// TIA Portal project "EMS" (V14)

(* hardware
DEVICE "S7-1200 station_2"  S7-1200 Station
   slot 0: "Rack_0"  S7-1200 Rack  Rack  V1.0
   slot 1: "EnergyManagement"  CPU 1211C AC/DC/Rly  6ES7 211-1BE40-0XB0  V4.2
   slot 101: "CM 1241 (RS422/485)_1"  6ES7 241-1CH32-0XB0  V2.2
*)

// ===== PLC "EnergyManagement"  CPU 1211C AC/DC/Rly =====

VAR_GLOBAL   // PLC tag table "Default tag table"
   "System_Byte" AT %MB1 : Byte;
   "FirstScan" AT %M1.0 : Bool;
   "DiagStatusUpdate" AT %M1.1 : Bool;
   "AlwaysTRUE" AT %M1.2 : Bool;
   "AlwaysFALSE" AT %M1.3 : Bool;
   "Clock_Byte" AT %MB0 : Byte;
   "Clock_10Hz" AT %M0.0 : Bool;
   "Clock_5Hz" AT %M0.1 : Bool;
   "Clock_2.5Hz" AT %M0.2 : Bool;
   "Clock_2Hz" AT %M0.3 : Bool;
   "Clock_1.25Hz" AT %M0.4 : Bool;
   "Clock_1Hz" AT %M0.5 : Bool;
   "Clock_0.625Hz" AT %M0.6 : Bool;
   "Clock_0.5Hz" AT %M0.7 : Bool;
   "Tag_1" AT %MB3 : Byte;
   "Tag_2" AT %M4.0 : Bool;
   "Tag_3" AT %M4.1 : Bool;
   "Tag_4" AT %M4.3 : Bool;
   "Tag_5" AT %M4.2 : Bool;
   "Tag_6" AT %MW102 : Word;
   "Tag_7" AT %M2.0 : Bool;
   "Tag_8" AT %M3.1 : Bool;
   "Tag_9" AT %MW10 : Word;
   "Tag_10" AT %MW100 : Word;
   "Tag_11" AT %M3.0 : Bool;
   "g" AT %M4.4 : Bool;
END_VAR

VAR_GLOBAL   // PLC tag table "GTL"
   "reteaOut" AT %Q0.0 : Bool;
   "baterieOut" AT %Q0.1 : Bool;
   "SPARE_OUT" AT %Q0.2 : Bool;
   "SPARE_OUT(1)" AT %Q0.3 : Bool;
   "stare" AT %I0.0 : Bool;
   "manual" AT %I0.2 : Bool;
   "retea" AT %I0.3 : Bool;
   "baterie" AT %I0.4 : Bool;
   "directieAuto" AT %I0.5 : Bool;   // FALSE - IntervalOrar TRUE - Piata
   "I1" AT %IW64 : Int;
   "I2" AT %IW66 : Int;
   "auto" AT %I0.1 : Bool;
END_VAR

VAR_GLOBAL CONSTANT   // PLC tag table "GTL"
   "Verificare" : Bool := 0;
END_VAR

TYPE "Modbus_Data"
   STRUCT
      Modbus : Struct
         Holding_Register : Struct
            Read : "UDT_DATA_PTR";
            Write : "UDT_DATA_PTR";
         END_STRUCT;
      END_STRUCT;
   END_STRUCT;
END_TYPE

TYPE "UDT_DATA_PTR"
   STRUCT
      DATA : Array[1..50] of Word;
   END_STRUCT;
END_TYPE

TYPE "UDT_MB_COMM_LOAD"
   STRUCT
      DONE : Bool;
      ERROR : Bool;
      STATUS : Word;
      ERROR_STATUS : Word;
   END_STRUCT;
END_TYPE

TYPE "Modbus_Slave_Data"
   STRUCT
      NDR : Bool;
      DR : Bool;
      ERROR : Bool;
      STATUS : Word;
      ERROR_STATUS : Word;
      MB_ADDR : UInt;
   END_STRUCT;
END_TYPE

TYPE "Modbus_M aster_Data"
   STRUCT
      DONE : Bool;
      BUSY : Bool;
      ERROR : Bool;
      STATUS : Word;
   END_STRUCT;
END_TYPE

DATA_BLOCK "GVL"   // DB3
{ S7_Optimized_Access := 'TRUE' }
VERSION : 0.1
   VAR
      "STEP" : Array[0..8] of Bool;
      MB_STEP : Array[0..8] of Bool;
   END_VAR
BEGIN
   "STEP"[0] := true;
   MB_STEP[0] := true;
END_DATA_BLOCK

DATA_BLOCK "IntervalOrar"   // DB6
{ S7_Optimized_Access := 'TRUE' }
VERSION : 0.1
   VAR
      "Error Code" : Word;
      OraCurenta : DTL;
      InceputProgram : DTL := DTL#1970-01-01-06:00:00;
      SfarsitProgram : DTL := DTL#1970-01-01-17:00:00;
   END_VAR
BEGIN
END_DATA_BLOCK

DATA_BLOCK "Piata"   // DB11
{ S7_Optimized_Access := 'TRUE' }
VERSION : 0.1
   VAR
      Prag : Int := 500;
      PretPiata : Int := 400;
   END_VAR
BEGIN
END_DATA_BLOCK

DATA_BLOCK "MB_Config"   // DB17
{ S7_Optimized_Access := 'FALSE' }
VERSION : 0.1
   VAR
      Modbus_Data : Struct
         DATA : Array[0..9] of UInt;
      END_STRUCT;
      Modbus_Data_1 : Struct
         DATA : Array[0..20] of Bool;
      END_STRUCT;
      Modbus_Slave : "Modbus_Slave_Data";
      MB_COMM_LOAD : "UDT_MB_COMM_LOAD";
      Modbus_Master : "Modbus_M aster_Data";
   END_VAR
BEGIN
   Modbus_Slave.MB_ADDR := 2;
   Modbus_Data.DATA[0] := 1;
   Modbus_Data.DATA[1] := 2;
   Modbus_Data.DATA[2] := 3;
   Modbus_Data.DATA[3] := 4;
   Modbus_Data.DATA[4] := 5;
   Modbus_Data.DATA[5] := 6;
   Modbus_Data.DATA[6] := 7;
   Modbus_Data.DATA[7] := 8;
   Modbus_Data.DATA[8] := 9;
END_DATA_BLOCK

DATA_BLOCK "ModBus_Commands"   // DB20
{ S7_Optimized_Access := 'FALSE' }
VERSION : 0.1
   VAR
      VERIF_REQUEST : Struct
         DATA : Array[1..8] of Byte;
      END_STRUCT;
      RESET_REQUEST : Struct
         DATA : Array[1..8] of Byte;
      END_STRUCT;
      SET_RETEA_ON : Struct   // DE VERIFICAT!! 42044
         DATA : Array[1..8] of Byte;
      END_STRUCT;
      SET_RETEA_OFF : Struct   // DE VERIFICAT!! 42044
         DATA : Array[1..8] of Byte;   // DE VERIFICAT!!
      END_STRUCT;
      SET_STARE_ON : Struct   // DE VERIFICAT!! 40200
         DATA : Array[1..8] of Byte;
      END_STRUCT;
      SET_STARE_OFF : Struct   // DE VERIFICAT!! 40200
         DATA : Array[1..8] of Byte;
      END_STRUCT;
      GET_CURR_HOUR_YIELD : Struct
         DATA : Array[1..8] of Byte;
      END_STRUCT;
      GET_CURR_DAY_YIELD : Struct
         DATA : Array[1..8] of Byte;
      END_STRUCT;
      GET_CURR_MONTH_YIELD : Struct
         DATA : Array[1..8] of Byte;
      END_STRUCT;
      GET_POWER_DIRECTION : Struct
         DATA : Array[1..8] of Byte;
      END_STRUCT;
      GET_DEVICE_STATUS : Struct
         DATA : Array[1..8] of Byte;
      END_STRUCT;
      PLACE_HOLDER : Struct
         DATA : Array[1..8] of Byte;
      END_STRUCT;
   END_VAR
BEGIN
   SET_RETEA_ON.DATA[8] := 16#68;
   SET_RETEA_ON.DATA[7] := 16#26;
   SET_RETEA_ON.DATA[6] := 16#01;
   SET_RETEA_ON.DATA[5] := 16#00;
   SET_RETEA_ON.DATA[4] := 16#34;
   SET_RETEA_ON.DATA[3] := 16#9D;
   SET_RETEA_ON.DATA[2] := 16#06;
   SET_RETEA_ON.DATA[1] := 16#01;
   SET_STARE_ON.DATA[8] := 16#64;
   SET_STARE_ON.DATA[7] := 16#E6;
   SET_STARE_ON.DATA[6] := 16#01;
   SET_STARE_ON.DATA[5] := 16#00;
   SET_STARE_ON.DATA[4] := 16#08;
   SET_STARE_ON.DATA[3] := 16#9D;
   SET_STARE_ON.DATA[2] := 16#06;
   SET_STARE_ON.DATA[1] := 16#01;
   RESET_REQUEST.DATA[1] := 16#FF;
   RESET_REQUEST.DATA[2] := 16#FF;
   RESET_REQUEST.DATA[3] := 16#FF;
   RESET_REQUEST.DATA[4] := 16#FF;
   RESET_REQUEST.DATA[5] := 16#FF;
   RESET_REQUEST.DATA[6] := 16#FF;
   RESET_REQUEST.DATA[7] := 16#FF;
   RESET_REQUEST.DATA[8] := 16#FF;
   GET_CURR_HOUR_YIELD.DATA[1] := 16#01;
   GET_CURR_HOUR_YIELD.DATA[2] := 16#03;
   GET_CURR_HOUR_YIELD.DATA[3] := 16#7D;
   GET_CURR_HOUR_YIELD.DATA[4] := 16#9E;
   GET_CURR_HOUR_YIELD.DATA[5] := 16#00;
   GET_CURR_HOUR_YIELD.DATA[6] := 16#02;
   GET_CURR_HOUR_YIELD.DATA[7] := 16#BD;
   GET_CURR_HOUR_YIELD.DATA[8] := 16#89;
   GET_CURR_DAY_YIELD.DATA[1] := 16#01;
   GET_CURR_DAY_YIELD.DATA[2] := 16#03;
   GET_CURR_DAY_YIELD.DATA[3] := 16#7D;
   GET_CURR_DAY_YIELD.DATA[4] := 16#A2;
   GET_CURR_DAY_YIELD.DATA[5] := 16#00;
   GET_CURR_DAY_YIELD.DATA[6] := 16#02;
   GET_CURR_DAY_YIELD.DATA[7] := 16#7D;
   GET_CURR_DAY_YIELD.DATA[8] := 16#85;
   GET_POWER_DIRECTION.DATA[8] := 16#3A;
   GET_POWER_DIRECTION.DATA[7] := 16#39;
   GET_POWER_DIRECTION.DATA[6] := 16#02;
   GET_POWER_DIRECTION.DATA[5] := 16#00;
   GET_POWER_DIRECTION.DATA[4] := 16#F9;
   GET_POWER_DIRECTION.DATA[3] := 16#90;
   GET_POWER_DIRECTION.DATA[2] := 16#03;
   GET_POWER_DIRECTION.DATA[1] := 16#01;
   SET_STARE_OFF.DATA[1] := 16#01;
   SET_STARE_OFF.DATA[2] := 16#06;
   SET_STARE_OFF.DATA[3] := 16#9D;
   SET_STARE_OFF.DATA[4] := 16#08;
   SET_STARE_OFF.DATA[5] := 16#00;
   SET_STARE_OFF.DATA[6] := 16#00;
   SET_STARE_OFF.DATA[7] := 16#27;
   SET_STARE_OFF.DATA[8] := 16#A2;
   SET_RETEA_OFF.DATA[1] := 16#01;
   SET_RETEA_OFF.DATA[2] := 16#06;
   SET_RETEA_OFF.DATA[3] := 16#9D;
   SET_RETEA_OFF.DATA[4] := 16#34;
   SET_RETEA_OFF.DATA[5] := 16#00;
   SET_RETEA_OFF.DATA[6] := 16#00;
   SET_RETEA_OFF.DATA[7] := 16#E7;
   SET_RETEA_OFF.DATA[8] := 16#A8;
   PLACE_HOLDER.DATA[1] := 16#FF;
   PLACE_HOLDER.DATA[2] := 16#FF;
   PLACE_HOLDER.DATA[3] := 16#FF;
   PLACE_HOLDER.DATA[4] := 16#FF;
   PLACE_HOLDER.DATA[5] := 16#FF;
   PLACE_HOLDER.DATA[6] := 16#FF;
   PLACE_HOLDER.DATA[7] := 16#FF;
   PLACE_HOLDER.DATA[8] := 16#FF;
   VERIF_REQUEST.DATA[1] := 16#01;
   VERIF_REQUEST.DATA[2] := 16#03;
   VERIF_REQUEST.DATA[3] := 16#FF;
   VERIF_REQUEST.DATA[4] := 16#FF;
   VERIF_REQUEST.DATA[5] := 16#FF;
   VERIF_REQUEST.DATA[6] := 16#FF;
   VERIF_REQUEST.DATA[7] := 16#FF;
   VERIF_REQUEST.DATA[8] := 16#FF;
   GET_DEVICE_STATUS.DATA[1] := 16#01;
   GET_DEVICE_STATUS.DATA[2] := 16#03;
   GET_DEVICE_STATUS.DATA[3] := 16#7D;
   GET_DEVICE_STATUS.DATA[4] := 16#59;
   GET_DEVICE_STATUS.DATA[5] := 16#00;
   GET_DEVICE_STATUS.DATA[6] := 16#01;
   GET_DEVICE_STATUS.DATA[7] := 16#4C;
   GET_DEVICE_STATUS.DATA[8] := 16#75;
   GET_CURR_MONTH_YIELD.DATA[1] := 16#01;
   GET_CURR_MONTH_YIELD.DATA[2] := 16#03;
   GET_CURR_MONTH_YIELD.DATA[3] := 16#7D;
   GET_CURR_MONTH_YIELD.DATA[4] := 16#76;
   GET_CURR_MONTH_YIELD.DATA[5] := 16#00;
   GET_CURR_MONTH_YIELD.DATA[6] := 16#02;
   GET_CURR_MONTH_YIELD.DATA[7] := 16#3D;
   GET_CURR_MONTH_YIELD.DATA[8] := 16#BD;
END_DATA_BLOCK

DATA_BLOCK "CUSTOM_MODBUS_CONFIG"   // DB21
{ S7_Optimized_Access := 'FALSE' }
VERSION : 0.1
   VAR
      Modbus_Data_BUFFER : Struct
         DATA : Array[1..40] of Byte;
      END_STRUCT;
      REQ_RESP : Struct
         DATA : Array[1..40] of Byte;
      END_STRUCT;
      SEND_REQUEST_BUFFER : Struct
         DATA : Array[1..8] of Byte;
      END_STRUCT;
      PORT_CONFIG : "UDT_MB_COMM_LOAD";
      PTP_CONFIG : Struct
         DONE : Bool;
         BUSY : Bool;
         ERROR : Bool;
         STATUS : Word;
         LENGTH : UInt := 8;
      END_STRUCT;
      RCV_CONFIG : Struct
         NDR : Bool;
         BUSY : Bool;
         ERROR : Bool;
         STATUS : Word;
         LENGTH : UInt;
      END_STRUCT;
      PULSE_GET_COUNTER : Int := 0;
      PULSE_GET_RESET : Bool := false;
      PULSE_GET_MOD : Int := 0;
      PULSE_SET_COUNTER : Int := 0;
      PULSE_SET_RESET : Bool := false;
      PULSE_SET_MOD : Int := 0;
      SECOND_COUNTER : Int := 0;
      SECOND_RESET : Bool := false;
      SECOND_MOD : Int := 0;
      CRC : Word := 16#FFFF;
      isValid : Bool;
      REQ_PULSE : Int;
      REQ_CLOCK : Bool;
      TEST_ONLY_OUT : Int;
   END_VAR
BEGIN
   Modbus_Data_BUFFER.DATA[2] := 16#0;
   Modbus_Data_BUFFER.DATA[1] := 16#0;
   Modbus_Data_BUFFER.DATA[8] := 16#0;
   Modbus_Data_BUFFER.DATA[7] := 16#0;
   Modbus_Data_BUFFER.DATA[5] := 16#0;
   Modbus_Data_BUFFER.DATA[6] := 16#0;
   Modbus_Data_BUFFER.DATA[4] := 16#0;
   Modbus_Data_BUFFER.DATA[3] := 16#0;
   SEND_REQUEST_BUFFER.DATA[1] := 16#FF;
   SEND_REQUEST_BUFFER.DATA[2] := 16#FF;
   SEND_REQUEST_BUFFER.DATA[3] := 16#FF;
   SEND_REQUEST_BUFFER.DATA[4] := 16#FF;
   SEND_REQUEST_BUFFER.DATA[5] := 16#FF;
   SEND_REQUEST_BUFFER.DATA[6] := 16#FF;
   SEND_REQUEST_BUFFER.DATA[7] := 16#FF;
   SEND_REQUEST_BUFFER.DATA[8] := 16#FF;
   Modbus_Data_BUFFER.DATA[9] := 16#0;
END_DATA_BLOCK

DATA_BLOCK "ModBus_Responses"   // DB27
{ S7_Optimized_Access := 'FALSE' }
VERSION : 0.1
   VAR
      CURR_HOUR_YIELD_RESPONSE : Struct
         DATA : Array[1..40] of Byte;
      END_STRUCT;
      CURR_DAY_YIELD_RESPONSE : Struct
         DATA : Array[1..40] of Byte;
      END_STRUCT;
      CURR_MONTH_YIELD_RESPONSE : Struct
         DATA : Array[1..40] of Byte;
      END_STRUCT;
      POWER_DIRECTION_RESPONSE : Struct
         DATA : Array[1..40] of Byte;
      END_STRUCT;
      DEVICE_STATUS_RESPONSE : Struct
         DATA : Array[1..40] of Byte;
      END_STRUCT;
      SET_STARE_RESPONSE : Struct
         DATA : Array[1..40] of Byte;
      END_STRUCT;
      TEST_ONLY : Struct
         DATA : Array[1..40] of Byte;
      END_STRUCT;
      TEST_ONLY_2 : Struct
         DATA : Array[1..40] of Byte;
      END_STRUCT;
   END_VAR
BEGIN
   TEST_ONLY_2.DATA[1] := 16#01;
   TEST_ONLY_2.DATA[2] := 16#03;
   TEST_ONLY_2.DATA[3] := 16#7D;
   TEST_ONLY_2.DATA[4] := 16#9E;
   TEST_ONLY_2.DATA[5] := 16#00;
   TEST_ONLY_2.DATA[6] := 16#02;
   TEST_ONLY_2.DATA[7] := 16#BD;
   TEST_ONLY_2.DATA[8] := 16#89;
END_DATA_BLOCK

DATA_BLOCK "DATA_INTERPRETATION"   // DB31
{ S7_Optimized_Access := 'TRUE' }
VERSION : 0.1
   VAR
      TEST_ONLY : DWord;
   END_VAR
BEGIN
END_DATA_BLOCK

DATA_BLOCK "READY_TO_SEND"   // DB33
{ S7_Optimized_Access := 'FALSE' }
VERSION : 0.1
   VAR
      just_started : Bool;
      CURR_HOUR_YIELD_RESPONSE : DInt;
      CURR_DAY_YIELD_RESPONSE : DInt;
      CURR_MONTH_YIELD_RESPONSE : DInt;
      POWER_DIRECTION_RESPONSE : DInt;
      DEVICE_STATUS_RESPONSE : DInt;
   END_VAR
BEGIN
END_DATA_BLOCK

// folder: System blocks/Program resources

DATA_BLOCK "IEC_Counter_0_DB"   // DB13
{ S7_Optimized_Access := 'TRUE' }
AUTHOR : Simatic
FAMILY : IEC
NAME : CNTR
VERSION : 1.0
// stored: InstanceOfName IEC_COUNTER
"IEC_COUNTER"
BEGIN
END_DATA_BLOCK

DATA_BLOCK "PULSE_GENERATOR_SET"   // DB26
{ S7_Optimized_Access := 'TRUE' }
AUTHOR : Simatic
FAMILY : IEC
NAME : CNTR
VERSION : 1.0
// stored: InstanceOfName IEC_COUNTER
"IEC_COUNTER"
BEGIN
END_DATA_BLOCK

DATA_BLOCK "PULSE_GENERATOR_GET"   // DB30
{ S7_Optimized_Access := 'TRUE' }
AUTHOR : Simatic
FAMILY : IEC
NAME : CNTR
VERSION : 1.0
// stored: InstanceOfName IEC_COUNTER
"IEC_COUNTER"
BEGIN
END_DATA_BLOCK

DATA_BLOCK "MINUTE_PULSE"   // DB32
{ S7_Optimized_Access := 'TRUE' }
AUTHOR : Simatic
FAMILY : IEC
NAME : CNTR
VERSION : 1.0
// stored: InstanceOfName IEC_COUNTER
"IEC_COUNTER"
BEGIN
END_DATA_BLOCK

// folder: (top level)

FUNCTION "MBus" : Void   // FC1, FBD
{ S7_Optimized_Access := 'TRUE' }
VERSION : 0.1
BEGIN

REGION Network 1
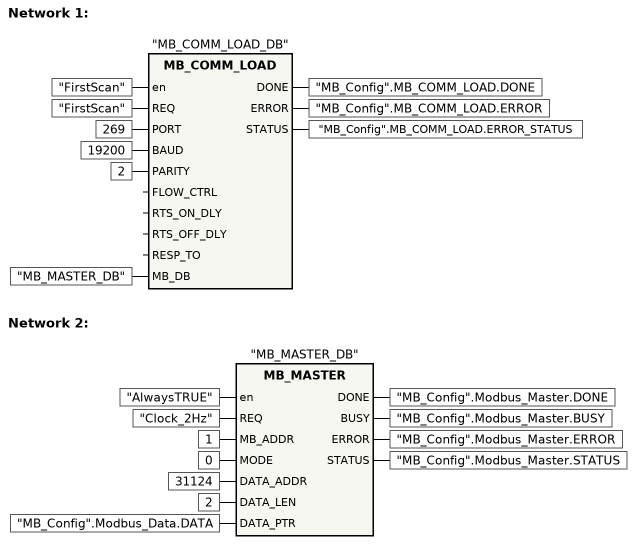
   IF "FirstScan" THEN
       "MB_COMM_LOAD_DB"(REQ := "FirstScan",   // MB_COMM_LOAD
                         PORT := 269,
                         BAUD := 19200,
                         PARITY := 2,
                         MB_DB := "MB_MASTER_DB",
                         DONE => "MB_Config".MB_COMM_LOAD.DONE,
                         ERROR => "MB_Config".MB_COMM_LOAD.ERROR,
                         STATUS => "MB_Config".MB_COMM_LOAD.ERROR_STATUS);
   END_IF;
END_REGION

REGION Network 2
   IF "AlwaysTRUE" THEN
       "MB_MASTER_DB"(REQ := "Clock_2Hz",   // MB_MASTER
                      MB_ADDR := 1,
                      MODE := 0,
                      DATA_ADDR := 31124,
                      DATA_LEN := 2,
                      DATA_PTR := "MB_Config".Modbus_Data.DATA,
                      DONE => "MB_Config".Modbus_Master.DONE,
                      BUSY => "MB_Config".Modbus_Master.BUSY,
                      ERROR => "MB_Config".Modbus_Master.ERROR,
                      STATUS => "MB_Config".Modbus_Master.STATUS);
   END_IF;
END_REGION
END_FUNCTION

FUNCTION "MBus_RTU" : Void   // FC2, FBD
{ S7_Optimized_Access := 'TRUE' }
VERSION : 0.1
BEGIN

REGION Network 1
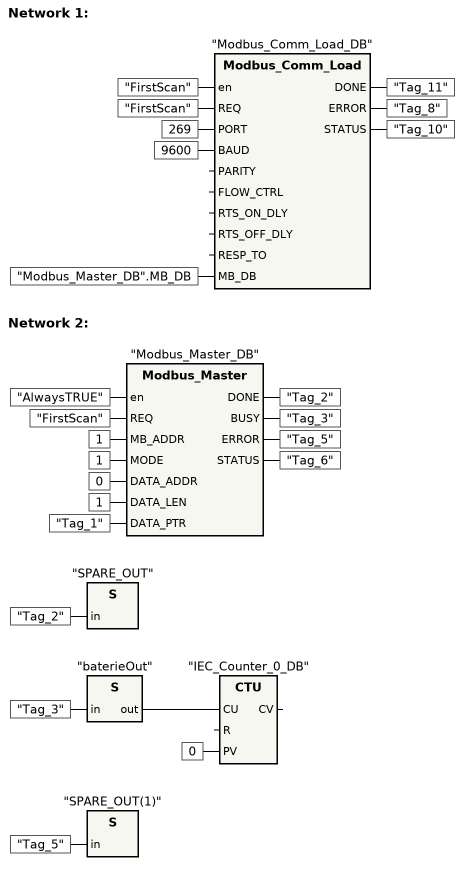
   IF "FirstScan" THEN
       "Modbus_Comm_Load_DB"(REQ := "FirstScan",   // Modbus_Comm_Load
                             PORT := 269,
                             BAUD := 9600,
                             MB_DB := "Modbus_Master_DB".MB_DB,
                             DONE => "Tag_11",
                             ERROR => "Tag_8",
                             STATUS => "Tag_10");
   END_IF;
END_REGION

REGION Network 2
   IF "AlwaysTRUE" THEN
       "Modbus_Master_DB"(REQ := "FirstScan",   // Modbus_Master
                          MB_ADDR := 1,
                          MODE := 1,
                          DATA_ADDR := 0,
                          DATA_LEN := 1,
                          DATA_PTR := "Tag_1",
                          DONE => "Tag_2",
                          BUSY => "Tag_3",
                          ERROR => "Tag_5",
                          STATUS => "Tag_6");
   END_IF;
   IF "Tag_2" THEN "SPARE_OUT" := TRUE; END_IF;
   IF "Tag_3" THEN "baterieOut" := TRUE; END_IF;
   "IEC_Counter_0_DB".CTU(CU := "Tag_3", PV := 0);
   IF "Tag_5" THEN "SPARE_OUT(1)" := TRUE; END_IF;
END_REGION
END_FUNCTION

FUNCTION "CUSTOM_MODBUS" : Void   // FC3, LAD
{ S7_Optimized_Access := 'TRUE' }
VERSION : 0.1
   VAR_INPUT
      COM : Struct
         DATA : Array[1..8] of Byte;
      END_STRUCT;
      PULSE : Bool;
   END_VAR
   VAR_IN_OUT
      BUFFER : Struct
         DATA : Array[1..40] of Byte;
      END_STRUCT;
   END_VAR
BEGIN

REGION Network 1
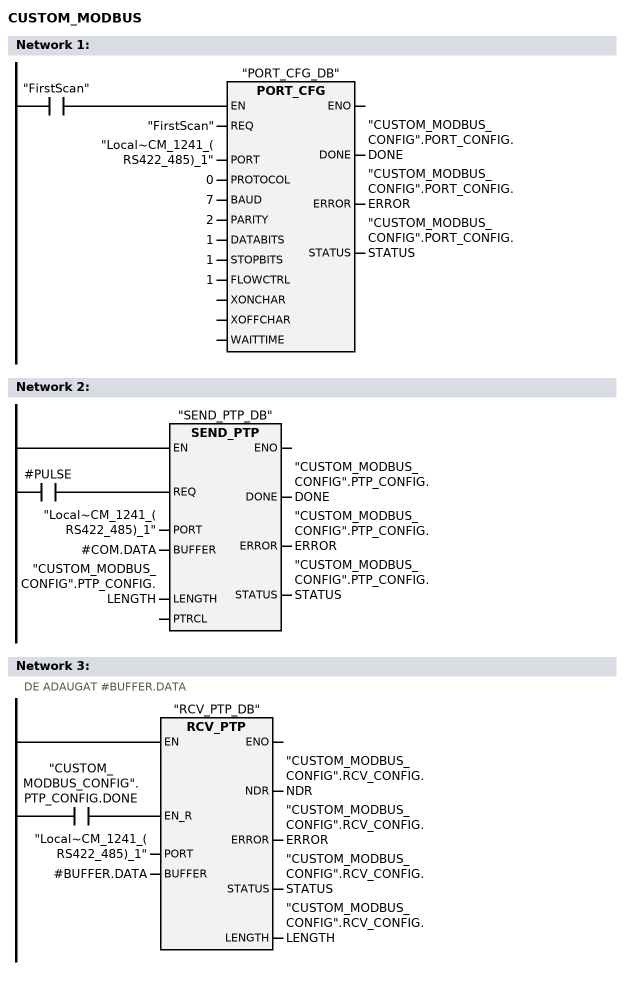
   IF "FirstScan" THEN
       "PORT_CFG_DB"(REQ := "FirstScan",   // PORT_CFG
                     PORT := "Local~CM_1241_(RS422_485)_1",
                     PROTOCOL := 0,
                     BAUD := 7,
                     PARITY := 2,
                     DATABITS := 1,
                     STOPBITS := 1,
                     FLOWCTRL := 1,
                     DONE => "CUSTOM_MODBUS_CONFIG".PORT_CONFIG.DONE,
                     ERROR => "CUSTOM_MODBUS_CONFIG".PORT_CONFIG.ERROR,
                     STATUS => "CUSTOM_MODBUS_CONFIG".PORT_CONFIG.STATUS);
   END_IF;
END_REGION

REGION Network 2
   "SEND_PTP_DB"(REQ := #PULSE,   // SEND_PTP
                 PORT := "Local~CM_1241_(RS422_485)_1",
                 BUFFER := #COM.DATA,
                 LENGTH := "CUSTOM_MODBUS_CONFIG".PTP_CONFIG.LENGTH,
                 DONE => "CUSTOM_MODBUS_CONFIG".PTP_CONFIG.DONE,
                 ERROR => "CUSTOM_MODBUS_CONFIG".PTP_CONFIG.ERROR,
                 STATUS => "CUSTOM_MODBUS_CONFIG".PTP_CONFIG.STATUS);
END_REGION

REGION Network 3
   // DE ADAUGAT #BUFFER.DATA
   "RCV_PTP_DB"(EN_R := "CUSTOM_MODBUS_CONFIG".PTP_CONFIG.DONE,   // RCV_PTP
                PORT := "Local~CM_1241_(RS422_485)_1",
                BUFFER := #BUFFER.DATA,
                NDR => "CUSTOM_MODBUS_CONFIG".RCV_CONFIG.NDR,
                ERROR => "CUSTOM_MODBUS_CONFIG".RCV_CONFIG.ERROR,
                STATUS => "CUSTOM_MODBUS_CONFIG".RCV_CONFIG.STATUS,
                LENGTH => "CUSTOM_MODBUS_CONFIG".RCV_CONFIG.LENGTH);
END_REGION
END_FUNCTION

FUNCTION "CRC" : Void   // FC4, SCL
{ S7_Optimized_Access := 'TRUE' }
VERSION : 0.1
   VAR_INPUT
      pData : Struct
         DATA : Array[1..40] of Byte;
      END_STRUCT;
      dLength : Int;
   END_VAR
   VAR_OUTPUT
      CRC : Word;   // Calculated CRC value
      out : Int;
      isCRCValid : Bool;
   END_VAR
   VAR_TEMP
      i : Int;   // Loop index for data bytes
      j : Int;   // Loop index for CRC bits
      iLength : Int;   // Number of bytes in the array
      bTemp : Byte;   // Temporary storage for byte data
      CRC_LSB : Bool;   // Least significant bit of CRC
      receivedCRC : Word;
   END_VAR
BEGIN
       // Initialize CRC to 0xFFFF
       #CRC:= 16#FFFF;

       #iLength := #dLength;
       IF #dLength = 0 THEN
           #iLength := 3 + #pData.DATA[3] + 2;
       END_IF;
       #out := #iLength - 2;



       // Calculate CRC for all bytes except the last two (CRC bytes)
       FOR #i := 1 TO (#iLength - 2) DO
           #bTemp := #pData.DATA[#i];
           #CRC := #CRC XOR BYTE_TO_WORD(#bTemp);

           // Process each bit in the byte
           FOR #j := 1 TO 8 DO
               #CRC_LSB := (#CRC AND 16#0001) <> 0; // Check the LSB of CRC
               #CRC := (#CRC / 2) AND 16#7FFF; // Logical right shift by 1 

               // If LSB was 1, XOR with the polynomial (0xA001)
               IF #CRC_LSB THEN
                   #CRC := #CRC XOR 16#A001;
               END_IF;
           END_FOR;
       END_FOR;

       // Retrieve the CRC from the last two bytes of input
       #receivedCRC := BYTE_TO_WORD(#pData.DATA[#iLength - 1]) + (BYTE_TO_WORD(#pData.DATA[#iLength]) * 256);

       // Compare calculated CRC with received CRC
       #isCRCValid := (#CRC = #receivedCRC);
END_FUNCTION

FUNCTION "Modbus_to_U32" : Void   // FC6, SCL
{ S7_Optimized_Access := 'TRUE' }
VERSION : 0.1
   VAR_INPUT
      pData : Struct
         DATA : Array[1..40] of Byte;
      END_STRUCT;
   END_VAR
   VAR_OUTPUT
      dataOut : DInt;
   END_VAR
   VAR_TEMP
      byteValue : Int;
      i : Int;
      iLength : Int;   // Number of bytes in the array
   END_VAR
BEGIN
   #iLength := #pData.DATA[3]; // Number of data bytes

   // Initialize the result
   #dataOut := 0;

   // Ensure dataLength is valid
   IF (#iLength > 0) AND (#iLength <= 4) THEN
       // Process each byte as a decimal digit
       FOR #i := 1 TO #iLength DO
           #byteValue :=BYTE_TO_DINT(#pData.DATA[3 + #i]); // Convert current byte to integer
           #dataOut := (#dataOut* 256) + #byteValue; // Treat as decimal and concatenate
       END_FOR;
   END_IF;
END_FUNCTION

ORGANIZATION_BLOCK "Main"   // OB1, LAD, ProgramCycle
TITLE = "Main Program Sweep (Cycle)"
{ S7_Optimized_Access := 'TRUE' }
VERSION : 0.1
   VAR_INPUT
      Initial_Call : Bool;   // Initial call of this OB
      Remanence : Bool;   // =True, if remanent data are available
   END_VAR
   VAR_TEMP   // added for the SCL form of the ladder/FBD networks
      _w1 : Bool;
   END_VAR
BEGIN

REGION Network 1: "R_TRIG_STEP1"
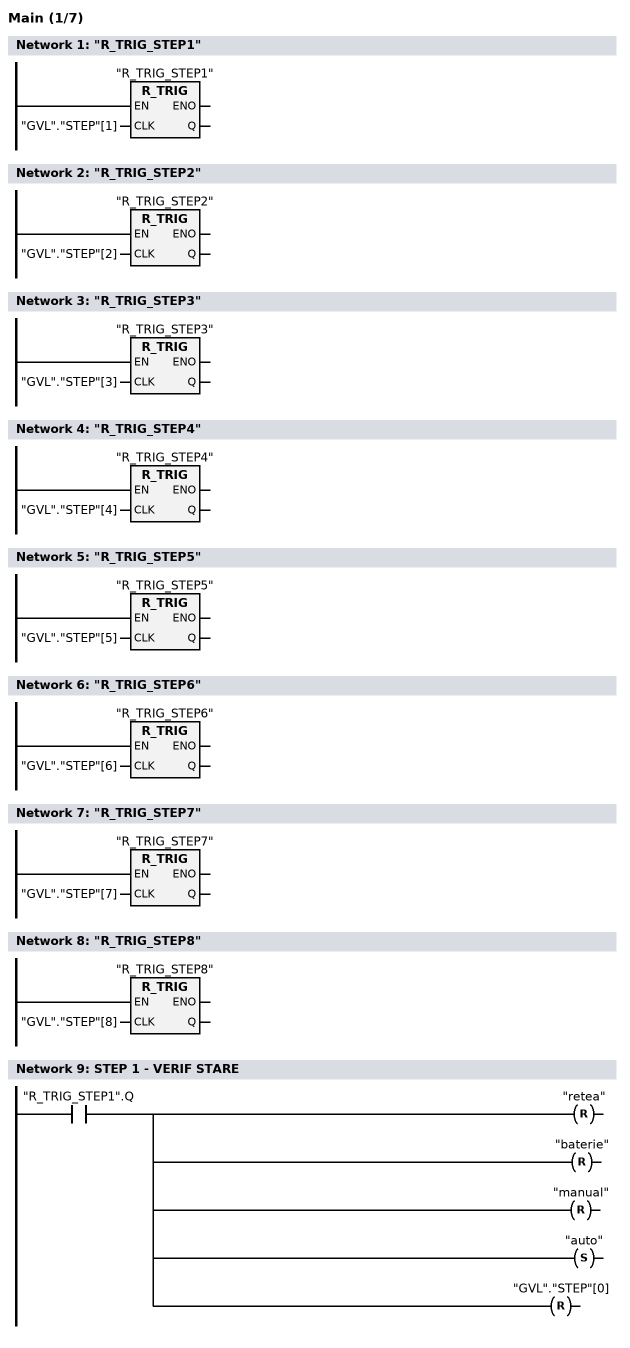
   "R_TRIG_STEP1"(CLK := "GVL"."STEP"[1]);   // R_TRIG
END_REGION

REGION Network 2: "R_TRIG_STEP2"
   "R_TRIG_STEP2"(CLK := "GVL"."STEP"[2]);   // R_TRIG
END_REGION

REGION Network 3: "R_TRIG_STEP3"
   "R_TRIG_STEP3"(CLK := "GVL"."STEP"[3]);   // R_TRIG
END_REGION

REGION Network 4: "R_TRIG_STEP4"
   "R_TRIG_STEP4"(CLK := "GVL"."STEP"[4]);   // R_TRIG
END_REGION

REGION Network 5: "R_TRIG_STEP5"
   "R_TRIG_STEP5"(CLK := "GVL"."STEP"[5]);   // R_TRIG
END_REGION

REGION Network 6: "R_TRIG_STEP6"
   "R_TRIG_STEP6"(CLK := "GVL"."STEP"[6]);   // R_TRIG
END_REGION

REGION Network 7: "R_TRIG_STEP7"
   "R_TRIG_STEP7"(CLK := "GVL"."STEP"[7]);   // R_TRIG
END_REGION

REGION Network 8: "R_TRIG_STEP8"
   "R_TRIG_STEP8"(CLK := "GVL"."STEP"[8]);   // R_TRIG
END_REGION

REGION Network 9: STEP 1 - VERIF STARE
   RUNG wire#powerrail
      Contact( "R_TRIG_STEP1".Q )
      wire#w1
      R_Coil( "retea" )
   END_RUNG
   RUNG wire#w1
      R_Coil( "baterie" )
   END_RUNG
   RUNG wire#w1
      R_Coil( "manual" )
   END_RUNG
   RUNG wire#w1
      S_Coil( "auto" )
   END_RUNG
   RUNG wire#w1
      R_Coil( "GVL"."STEP"[0] )
   END_RUNG
   // the same network as SCL:
   IF "R_TRIG_STEP1".Q THEN
       "retea" := FALSE;
       "baterie" := FALSE;
       "manual" := FALSE;
       "auto" := TRUE;
       "GVL"."STEP"[0] := FALSE;
   END_IF;
END_REGION

REGION Network 10: STEP 2 - MANUAL RETEA
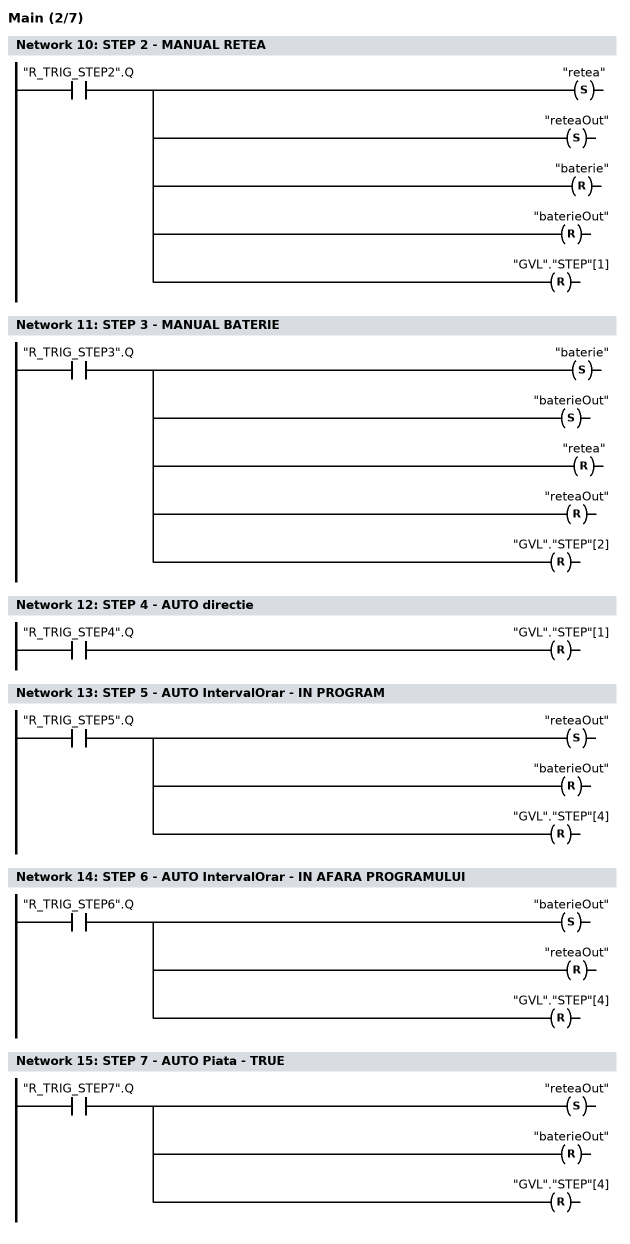
   RUNG wire#powerrail
      Contact( "R_TRIG_STEP2".Q )
      wire#w1
      S_Coil( "retea" )
   END_RUNG
   RUNG wire#w1
      S_Coil( "reteaOut" )
   END_RUNG
   RUNG wire#w1
      R_Coil( "baterie" )
   END_RUNG
   RUNG wire#w1
      R_Coil( "baterieOut" )
   END_RUNG
   RUNG wire#w1
      R_Coil( "GVL"."STEP"[1] )
   END_RUNG
   // the same network as SCL:
   IF "R_TRIG_STEP2".Q THEN
       "retea" := TRUE;
       "reteaOut" := TRUE;
       "baterie" := FALSE;
       "baterieOut" := FALSE;
       "GVL"."STEP"[1] := FALSE;
   END_IF;
END_REGION

REGION Network 11: STEP 3 - MANUAL BATERIE
   RUNG wire#powerrail
      Contact( "R_TRIG_STEP3".Q )
      wire#w1
      S_Coil( "baterie" )
   END_RUNG
   RUNG wire#w1
      S_Coil( "baterieOut" )
   END_RUNG
   RUNG wire#w1
      R_Coil( "retea" )
   END_RUNG
   RUNG wire#w1
      R_Coil( "reteaOut" )
   END_RUNG
   RUNG wire#w1
      R_Coil( "GVL"."STEP"[2] )
   END_RUNG
   // the same network as SCL:
   IF "R_TRIG_STEP3".Q THEN
       "baterie" := TRUE;
       "baterieOut" := TRUE;
       "retea" := FALSE;
       "reteaOut" := FALSE;
       "GVL"."STEP"[2] := FALSE;
   END_IF;
END_REGION

REGION Network 12: STEP 4 - AUTO directie
   RUNG wire#powerrail
      Contact( "R_TRIG_STEP4".Q )
      R_Coil( "GVL"."STEP"[1] )
   END_RUNG
   // the same network as SCL:
   IF "R_TRIG_STEP4".Q THEN "GVL"."STEP"[1] := FALSE; END_IF;
END_REGION

REGION Network 13: STEP 5 - AUTO IntervalOrar - IN PROGRAM
   RUNG wire#powerrail
      Contact( "R_TRIG_STEP5".Q )
      wire#w1
      S_Coil( "reteaOut" )
   END_RUNG
   RUNG wire#w1
      R_Coil( "baterieOut" )
   END_RUNG
   RUNG wire#w1
      R_Coil( "GVL"."STEP"[4] )
   END_RUNG
   // the same network as SCL:
   IF "R_TRIG_STEP5".Q THEN
       "reteaOut" := TRUE;
       "baterieOut" := FALSE;
       "GVL"."STEP"[4] := FALSE;
   END_IF;
END_REGION

REGION Network 14: STEP 6 - AUTO IntervalOrar - IN AFARA PROGRAMULUI
   RUNG wire#powerrail
      Contact( "R_TRIG_STEP6".Q )
      wire#w1
      S_Coil( "baterieOut" )
   END_RUNG
   RUNG wire#w1
      R_Coil( "reteaOut" )
   END_RUNG
   RUNG wire#w1
      R_Coil( "GVL"."STEP"[4] )
   END_RUNG
   // the same network as SCL:
   IF "R_TRIG_STEP6".Q THEN
       "baterieOut" := TRUE;
       "reteaOut" := FALSE;
       "GVL"."STEP"[4] := FALSE;
   END_IF;
END_REGION

REGION Network 15: STEP 7 - AUTO Piata - TRUE
   RUNG wire#powerrail
      Contact( "R_TRIG_STEP7".Q )
      wire#w1
      S_Coil( "reteaOut" )
   END_RUNG
   RUNG wire#w1
      R_Coil( "baterieOut" )
   END_RUNG
   RUNG wire#w1
      R_Coil( "GVL"."STEP"[4] )
   END_RUNG
   // the same network as SCL:
   IF "R_TRIG_STEP7".Q THEN
       "reteaOut" := TRUE;
       "baterieOut" := FALSE;
       "GVL"."STEP"[4] := FALSE;
   END_IF;
END_REGION

REGION Network 16: STEP 8 - AUTO Piata - FALSE
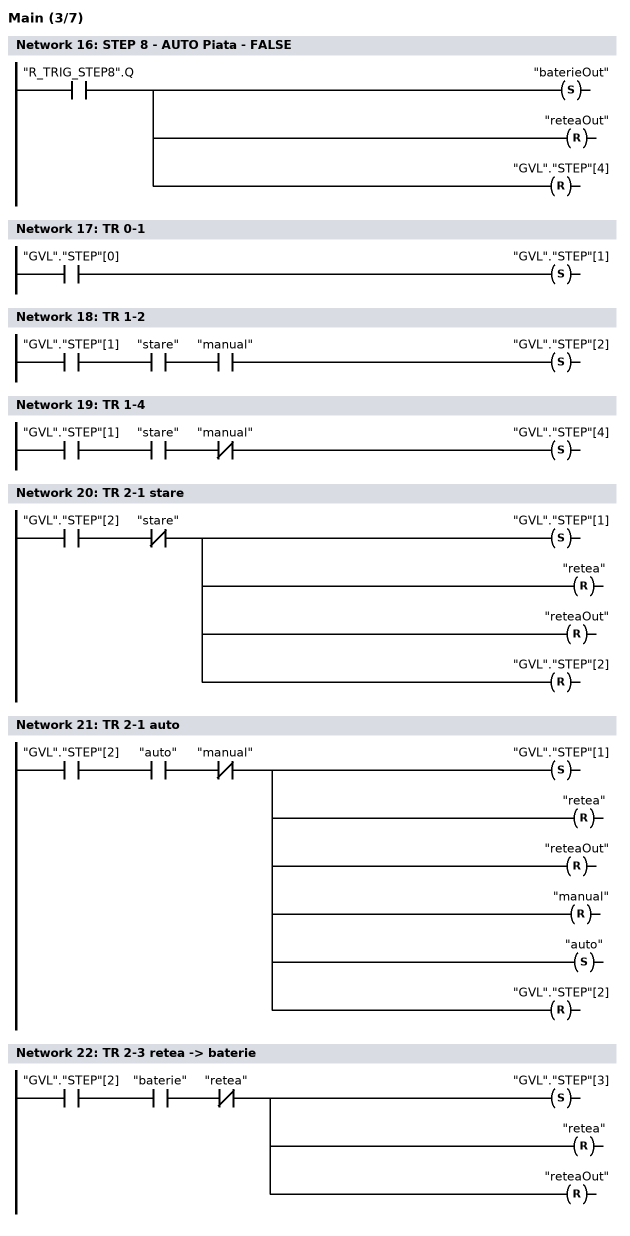
   RUNG wire#powerrail
      Contact( "R_TRIG_STEP8".Q )
      wire#w1
      S_Coil( "baterieOut" )
   END_RUNG
   RUNG wire#w1
      R_Coil( "reteaOut" )
   END_RUNG
   RUNG wire#w1
      R_Coil( "GVL"."STEP"[4] )
   END_RUNG
   // the same network as SCL:
   IF "R_TRIG_STEP8".Q THEN
       "baterieOut" := TRUE;
       "reteaOut" := FALSE;
       "GVL"."STEP"[4] := FALSE;
   END_IF;
END_REGION

REGION Network 17: TR 0-1
   RUNG wire#powerrail
      Contact( "GVL"."STEP"[0] )
      S_Coil( "GVL"."STEP"[1] )
   END_RUNG
   // the same network as SCL:
   IF "GVL"."STEP"[0] THEN "GVL"."STEP"[1] := TRUE; END_IF;
END_REGION

REGION Network 18: TR 1-2
   RUNG wire#powerrail
      Contact( "GVL"."STEP"[1] )
      Contact( "stare" )
      Contact( "manual" )
      S_Coil( "GVL"."STEP"[2] )
   END_RUNG
   // the same network as SCL:
   IF "GVL"."STEP"[1] AND "stare" AND "manual" THEN "GVL"."STEP"[2] := TRUE; END_IF;
END_REGION

REGION Network 19: TR 1-4
   RUNG wire#powerrail
      Contact( "GVL"."STEP"[1] )
      Contact( "stare" )
      I_Contact( "manual" )
      S_Coil( "GVL"."STEP"[4] )
   END_RUNG
   // the same network as SCL:
   IF "GVL"."STEP"[1] AND "stare" AND NOT "manual" THEN "GVL"."STEP"[4] := TRUE; END_IF;
END_REGION

REGION Network 20: TR 2-1 stare
   RUNG wire#powerrail
      Contact( "GVL"."STEP"[2] )
      I_Contact( "stare" )
      wire#w1
      S_Coil( "GVL"."STEP"[1] )
   END_RUNG
   RUNG wire#w1
      R_Coil( "retea" )
   END_RUNG
   RUNG wire#w1
      R_Coil( "reteaOut" )
   END_RUNG
   RUNG wire#w1
      R_Coil( "GVL"."STEP"[2] )
   END_RUNG
   // the same network as SCL:
   #_w1 := "GVL"."STEP"[2] AND NOT "stare";
   IF #_w1 THEN
       "GVL"."STEP"[1] := TRUE;
       "retea" := FALSE;
       "reteaOut" := FALSE;
       "GVL"."STEP"[2] := FALSE;
   END_IF;
END_REGION

REGION Network 21: TR 2-1 auto
   RUNG wire#powerrail
      Contact( "GVL"."STEP"[2] )
      Contact( "auto" )
      I_Contact( "manual" )
      wire#w1
      S_Coil( "GVL"."STEP"[1] )
   END_RUNG
   RUNG wire#w1
      R_Coil( "retea" )
   END_RUNG
   RUNG wire#w1
      R_Coil( "reteaOut" )
   END_RUNG
   RUNG wire#w1
      R_Coil( "manual" )
   END_RUNG
   RUNG wire#w1
      S_Coil( "auto" )
   END_RUNG
   RUNG wire#w1
      R_Coil( "GVL"."STEP"[2] )
   END_RUNG
   // the same network as SCL:
   #_w1 := "GVL"."STEP"[2] AND "auto" AND NOT "manual";
   IF #_w1 THEN
       "GVL"."STEP"[1] := TRUE;
       "retea" := FALSE;
       "reteaOut" := FALSE;
       "manual" := FALSE;
       "auto" := TRUE;
       "GVL"."STEP"[2] := FALSE;
   END_IF;
END_REGION

REGION Network 22: TR 2-3 retea -> baterie
   RUNG wire#powerrail
      Contact( "GVL"."STEP"[2] )
      Contact( "baterie" )
      I_Contact( "retea" )
      wire#w1
      S_Coil( "GVL"."STEP"[3] )
   END_RUNG
   RUNG wire#w1
      R_Coil( "retea" )
   END_RUNG
   RUNG wire#w1
      R_Coil( "reteaOut" )
   END_RUNG
   // the same network as SCL:
   #_w1 := "GVL"."STEP"[2] AND "baterie" AND NOT "retea";
   IF #_w1 THEN
       "GVL"."STEP"[3] := TRUE;
       "retea" := FALSE;
       "reteaOut" := FALSE;
   END_IF;
END_REGION

REGION Network 23: TR 3-1 stare
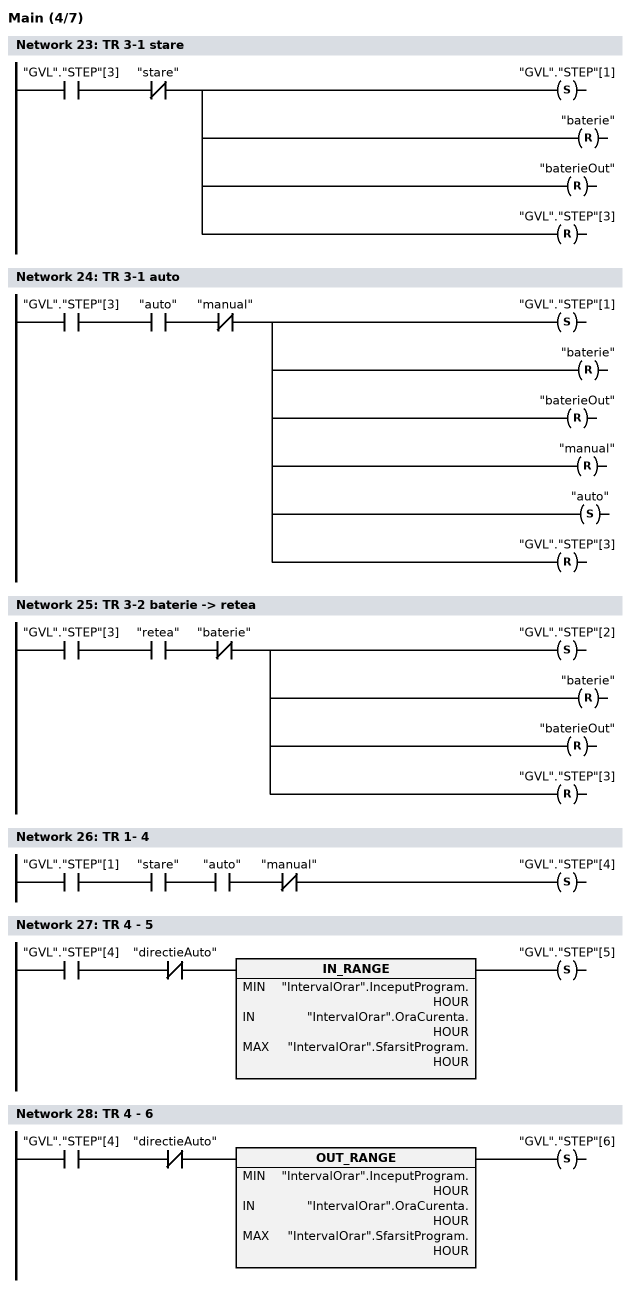
   RUNG wire#powerrail
      Contact( "GVL"."STEP"[3] )
      I_Contact( "stare" )
      wire#w1
      S_Coil( "GVL"."STEP"[1] )
   END_RUNG
   RUNG wire#w1
      R_Coil( "baterie" )
   END_RUNG
   RUNG wire#w1
      R_Coil( "baterieOut" )
   END_RUNG
   RUNG wire#w1
      R_Coil( "GVL"."STEP"[3] )
   END_RUNG
   // the same network as SCL:
   #_w1 := "GVL"."STEP"[3] AND NOT "stare";
   IF #_w1 THEN
       "GVL"."STEP"[1] := TRUE;
       "baterie" := FALSE;
       "baterieOut" := FALSE;
       "GVL"."STEP"[3] := FALSE;
   END_IF;
END_REGION

REGION Network 24: TR 3-1 auto
   RUNG wire#powerrail
      Contact( "GVL"."STEP"[3] )
      Contact( "auto" )
      I_Contact( "manual" )
      wire#w1
      S_Coil( "GVL"."STEP"[1] )
   END_RUNG
   RUNG wire#w1
      R_Coil( "baterie" )
   END_RUNG
   RUNG wire#w1
      R_Coil( "baterieOut" )
   END_RUNG
   RUNG wire#w1
      R_Coil( "manual" )
   END_RUNG
   RUNG wire#w1
      S_Coil( "auto" )
   END_RUNG
   RUNG wire#w1
      R_Coil( "GVL"."STEP"[3] )
   END_RUNG
   // the same network as SCL:
   #_w1 := "GVL"."STEP"[3] AND "auto" AND NOT "manual";
   IF #_w1 THEN
       "GVL"."STEP"[1] := TRUE;
       "baterie" := FALSE;
       "baterieOut" := FALSE;
       "manual" := FALSE;
       "auto" := TRUE;
       "GVL"."STEP"[3] := FALSE;
   END_IF;
END_REGION

REGION Network 25: TR 3-2 baterie -> retea
   RUNG wire#powerrail
      Contact( "GVL"."STEP"[3] )
      Contact( "retea" )
      I_Contact( "baterie" )
      wire#w1
      S_Coil( "GVL"."STEP"[2] )
   END_RUNG
   RUNG wire#w1
      R_Coil( "baterie" )
   END_RUNG
   RUNG wire#w1
      R_Coil( "baterieOut" )
   END_RUNG
   RUNG wire#w1
      R_Coil( "GVL"."STEP"[3] )
   END_RUNG
   // the same network as SCL:
   #_w1 := "GVL"."STEP"[3] AND "retea" AND NOT "baterie";
   IF #_w1 THEN
       "GVL"."STEP"[2] := TRUE;
       "baterie" := FALSE;
       "baterieOut" := FALSE;
       "GVL"."STEP"[3] := FALSE;
   END_IF;
END_REGION

REGION Network 26: TR 1- 4
   RUNG wire#powerrail
      Contact( "GVL"."STEP"[1] )
      Contact( "stare" )
      Contact( "auto" )
      I_Contact( "manual" )
      S_Coil( "GVL"."STEP"[4] )
   END_RUNG
   // the same network as SCL:
   IF "GVL"."STEP"[1] AND "stare" AND "auto" AND NOT "manual" THEN "GVL"."STEP"[4] := TRUE; END_IF;
END_REGION

REGION Network 27: TR 4 - 5
   RUNG wire#powerrail
      Contact( "GVL"."STEP"[4] )
      I_Contact( "directieAuto" )
      { S7_Templates := "SrcType := USInt" } InRange(min := "IntervalOrar".InceputProgram.HOUR, in := "IntervalOrar".OraCurenta.HOUR, max := "IntervalOrar".SfarsitProgram.HOUR)
      S_Coil( "GVL"."STEP"[5] )
   END_RUNG
   // the same network as SCL:
   IF "GVL"."STEP"[4] AND NOT "directieAuto" AND ("IntervalOrar".InceputProgram.HOUR <= "IntervalOrar".OraCurenta.HOUR) AND ("IntervalOrar".OraCurenta.HOUR <= "IntervalOrar".SfarsitProgram.HOUR) THEN
       "GVL"."STEP"[5] := TRUE;
   END_IF;
END_REGION

REGION Network 28: TR 4 - 6
   IF "GVL"."STEP"[4] AND NOT "directieAuto" AND (("IntervalOrar".OraCurenta.HOUR < "IntervalOrar".InceputProgram.HOUR) OR ("IntervalOrar".OraCurenta.HOUR > "IntervalOrar".SfarsitProgram.HOUR)) THEN
       "GVL"."STEP"[6] := TRUE;
   END_IF;
END_REGION

REGION Network 29: TR 4 - 7
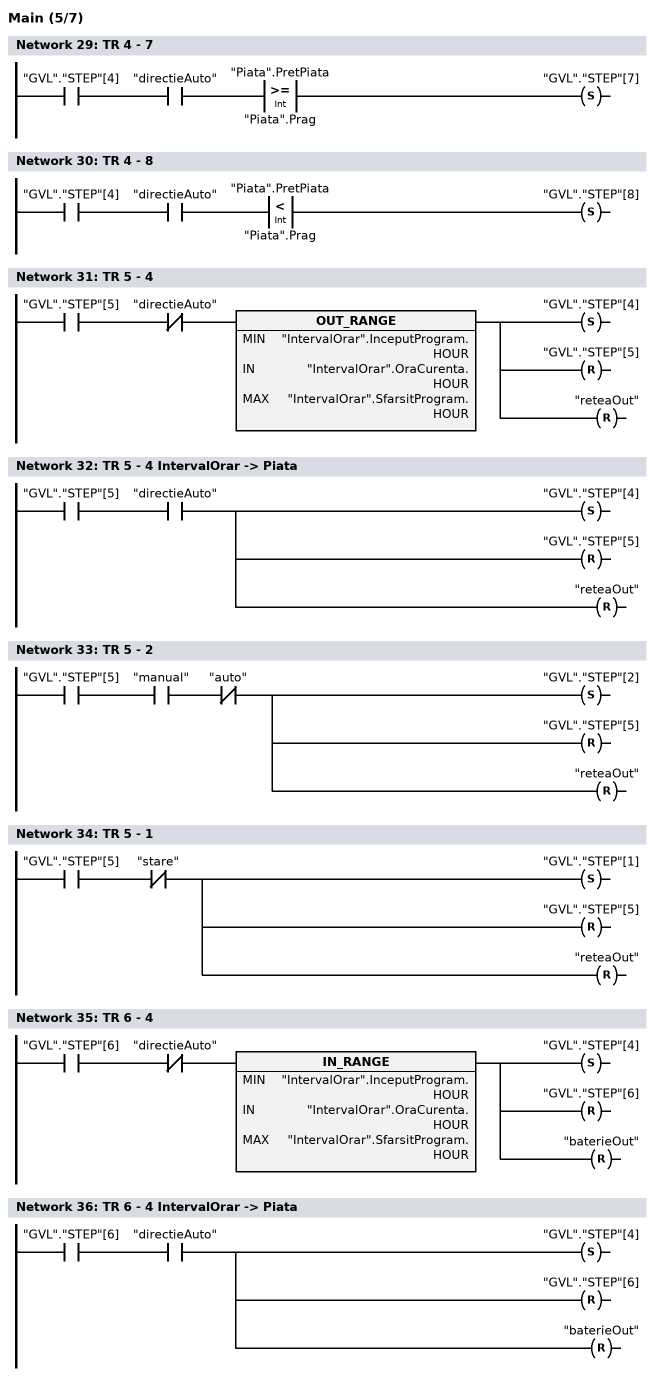
   RUNG wire#powerrail
      Contact( "GVL"."STEP"[4] )
      Contact( "directieAuto" )
      { S7_Templates := "SrcType := Int" } GE_Contact(in1 := "Piata".PretPiata, in2 := "Piata".Prag)
      S_Coil( "GVL"."STEP"[7] )
   END_RUNG
   // the same network as SCL:
   IF "GVL"."STEP"[4] AND "directieAuto" AND ("Piata".PretPiata >= "Piata".Prag) THEN
       "GVL"."STEP"[7] := TRUE;
   END_IF;
END_REGION

REGION Network 30: TR 4 - 8
   RUNG wire#powerrail
      Contact( "GVL"."STEP"[4] )
      Contact( "directieAuto" )
      { S7_Templates := "SrcType := Int" } LT_Contact(in1 := "Piata".PretPiata, in2 := "Piata".Prag)
      S_Coil( "GVL"."STEP"[8] )
   END_RUNG
   // the same network as SCL:
   IF "GVL"."STEP"[4] AND "directieAuto" AND ("Piata".PretPiata < "Piata".Prag) THEN
       "GVL"."STEP"[8] := TRUE;
   END_IF;
END_REGION

REGION Network 31: TR 5 - 4
   #_w1 := "GVL"."STEP"[5] AND NOT "directieAuto" AND (("IntervalOrar".OraCurenta.HOUR < "IntervalOrar".InceputProgram.HOUR) OR ("IntervalOrar".OraCurenta.HOUR > "IntervalOrar".SfarsitProgram.HOUR));
   IF #_w1 THEN
       "GVL"."STEP"[4] := TRUE;
       "GVL"."STEP"[5] := FALSE;
       "reteaOut" := FALSE;
   END_IF;
END_REGION

REGION Network 32: TR 5 - 4 IntervalOrar -> Piata
   RUNG wire#powerrail
      Contact( "GVL"."STEP"[5] )
      Contact( "directieAuto" )
      wire#w1
      S_Coil( "GVL"."STEP"[4] )
   END_RUNG
   RUNG wire#w1
      R_Coil( "GVL"."STEP"[5] )
   END_RUNG
   RUNG wire#w1
      R_Coil( "reteaOut" )
   END_RUNG
   // the same network as SCL:
   #_w1 := "GVL"."STEP"[5] AND "directieAuto";
   IF #_w1 THEN
       "GVL"."STEP"[4] := TRUE;
       "GVL"."STEP"[5] := FALSE;
       "reteaOut" := FALSE;
   END_IF;
END_REGION

REGION Network 33: TR 5 - 2
   RUNG wire#powerrail
      Contact( "GVL"."STEP"[5] )
      Contact( "manual" )
      I_Contact( "auto" )
      wire#w1
      S_Coil( "GVL"."STEP"[2] )
   END_RUNG
   RUNG wire#w1
      R_Coil( "GVL"."STEP"[5] )
   END_RUNG
   RUNG wire#w1
      R_Coil( "reteaOut" )
   END_RUNG
   // the same network as SCL:
   #_w1 := "GVL"."STEP"[5] AND "manual" AND NOT "auto";
   IF #_w1 THEN
       "GVL"."STEP"[2] := TRUE;
       "GVL"."STEP"[5] := FALSE;
       "reteaOut" := FALSE;
   END_IF;
END_REGION

REGION Network 34: TR 5 - 1
   RUNG wire#powerrail
      Contact( "GVL"."STEP"[5] )
      I_Contact( "stare" )
      wire#w1
      S_Coil( "GVL"."STEP"[1] )
   END_RUNG
   RUNG wire#w1
      R_Coil( "GVL"."STEP"[5] )
   END_RUNG
   RUNG wire#w1
      R_Coil( "reteaOut" )
   END_RUNG
   // the same network as SCL:
   #_w1 := "GVL"."STEP"[5] AND NOT "stare";
   IF #_w1 THEN
       "GVL"."STEP"[1] := TRUE;
       "GVL"."STEP"[5] := FALSE;
       "reteaOut" := FALSE;
   END_IF;
END_REGION

REGION Network 35: TR 6 - 4
   RUNG wire#powerrail
      Contact( "GVL"."STEP"[6] )
      I_Contact( "directieAuto" )
      { S7_Templates := "SrcType := USInt" } InRange(min := "IntervalOrar".InceputProgram.HOUR, in := "IntervalOrar".OraCurenta.HOUR, max := "IntervalOrar".SfarsitProgram.HOUR)
      wire#w1
      S_Coil( "GVL"."STEP"[4] )
   END_RUNG
   RUNG wire#w1
      R_Coil( "GVL"."STEP"[6] )
   END_RUNG
   RUNG wire#w1
      R_Coil( "baterieOut" )
   END_RUNG
   // the same network as SCL:
   #_w1 := "GVL"."STEP"[6] AND NOT "directieAuto" AND ("IntervalOrar".InceputProgram.HOUR <= "IntervalOrar".OraCurenta.HOUR) AND ("IntervalOrar".OraCurenta.HOUR <= "IntervalOrar".SfarsitProgram.HOUR);
   IF #_w1 THEN
       "GVL"."STEP"[4] := TRUE;
       "GVL"."STEP"[6] := FALSE;
       "baterieOut" := FALSE;
   END_IF;
END_REGION

REGION Network 36: TR 6 - 4 IntervalOrar -> Piata
   RUNG wire#powerrail
      Contact( "GVL"."STEP"[6] )
      Contact( "directieAuto" )
      wire#w1
      S_Coil( "GVL"."STEP"[4] )
   END_RUNG
   RUNG wire#w1
      R_Coil( "GVL"."STEP"[6] )
   END_RUNG
   RUNG wire#w1
      R_Coil( "baterieOut" )
   END_RUNG
   // the same network as SCL:
   #_w1 := "GVL"."STEP"[6] AND "directieAuto";
   IF #_w1 THEN
       "GVL"."STEP"[4] := TRUE;
       "GVL"."STEP"[6] := FALSE;
       "baterieOut" := FALSE;
   END_IF;
END_REGION

REGION Network 37: TR 6 - 2
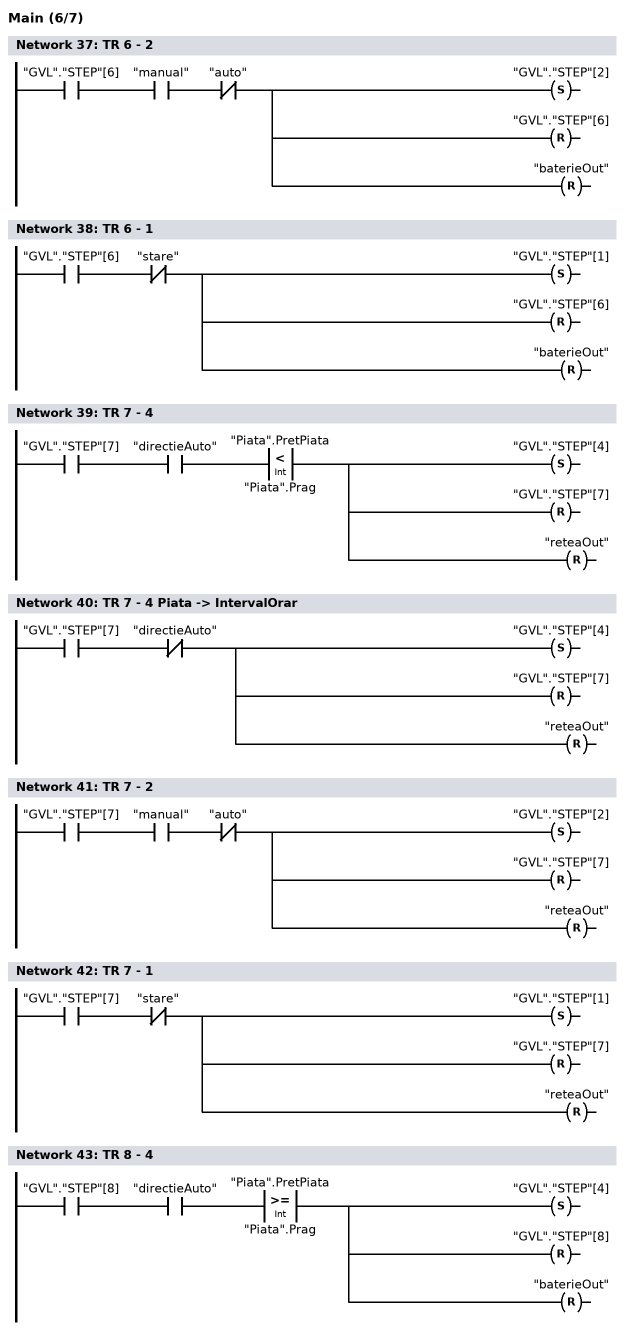
   RUNG wire#powerrail
      Contact( "GVL"."STEP"[6] )
      Contact( "manual" )
      I_Contact( "auto" )
      wire#w1
      S_Coil( "GVL"."STEP"[2] )
   END_RUNG
   RUNG wire#w1
      R_Coil( "GVL"."STEP"[6] )
   END_RUNG
   RUNG wire#w1
      R_Coil( "baterieOut" )
   END_RUNG
   // the same network as SCL:
   #_w1 := "GVL"."STEP"[6] AND "manual" AND NOT "auto";
   IF #_w1 THEN
       "GVL"."STEP"[2] := TRUE;
       "GVL"."STEP"[6] := FALSE;
       "baterieOut" := FALSE;
   END_IF;
END_REGION

REGION Network 38: TR 6 - 1
   RUNG wire#powerrail
      Contact( "GVL"."STEP"[6] )
      I_Contact( "stare" )
      wire#w1
      S_Coil( "GVL"."STEP"[1] )
   END_RUNG
   RUNG wire#w1
      R_Coil( "GVL"."STEP"[6] )
   END_RUNG
   RUNG wire#w1
      R_Coil( "baterieOut" )
   END_RUNG
   // the same network as SCL:
   #_w1 := "GVL"."STEP"[6] AND NOT "stare";
   IF #_w1 THEN
       "GVL"."STEP"[1] := TRUE;
       "GVL"."STEP"[6] := FALSE;
       "baterieOut" := FALSE;
   END_IF;
END_REGION

REGION Network 39: TR 7 - 4
   RUNG wire#powerrail
      Contact( "GVL"."STEP"[7] )
      Contact( "directieAuto" )
      { S7_Templates := "SrcType := Int" } LT_Contact(in1 := "Piata".PretPiata, in2 := "Piata".Prag)
      wire#w1
      S_Coil( "GVL"."STEP"[4] )
   END_RUNG
   RUNG wire#w1
      R_Coil( "GVL"."STEP"[7] )
   END_RUNG
   RUNG wire#w1
      R_Coil( "reteaOut" )
   END_RUNG
   // the same network as SCL:
   #_w1 := "GVL"."STEP"[7] AND "directieAuto" AND ("Piata".PretPiata < "Piata".Prag);
   IF #_w1 THEN
       "GVL"."STEP"[4] := TRUE;
       "GVL"."STEP"[7] := FALSE;
       "reteaOut" := FALSE;
   END_IF;
END_REGION

REGION Network 40: TR 7 - 4 Piata -> IntervalOrar
   RUNG wire#powerrail
      Contact( "GVL"."STEP"[7] )
      I_Contact( "directieAuto" )
      wire#w1
      S_Coil( "GVL"."STEP"[4] )
   END_RUNG
   RUNG wire#w1
      R_Coil( "GVL"."STEP"[7] )
   END_RUNG
   RUNG wire#w1
      R_Coil( "reteaOut" )
   END_RUNG
   // the same network as SCL:
   #_w1 := "GVL"."STEP"[7] AND NOT "directieAuto";
   IF #_w1 THEN
       "GVL"."STEP"[4] := TRUE;
       "GVL"."STEP"[7] := FALSE;
       "reteaOut" := FALSE;
   END_IF;
END_REGION

REGION Network 41: TR 7 - 2
   RUNG wire#powerrail
      Contact( "GVL"."STEP"[7] )
      Contact( "manual" )
      I_Contact( "auto" )
      wire#w1
      S_Coil( "GVL"."STEP"[2] )
   END_RUNG
   RUNG wire#w1
      R_Coil( "GVL"."STEP"[7] )
   END_RUNG
   RUNG wire#w1
      R_Coil( "reteaOut" )
   END_RUNG
   // the same network as SCL:
   #_w1 := "GVL"."STEP"[7] AND "manual" AND NOT "auto";
   IF #_w1 THEN
       "GVL"."STEP"[2] := TRUE;
       "GVL"."STEP"[7] := FALSE;
       "reteaOut" := FALSE;
   END_IF;
END_REGION

REGION Network 42: TR 7 - 1
   RUNG wire#powerrail
      Contact( "GVL"."STEP"[7] )
      I_Contact( "stare" )
      wire#w1
      S_Coil( "GVL"."STEP"[1] )
   END_RUNG
   RUNG wire#w1
      R_Coil( "GVL"."STEP"[7] )
   END_RUNG
   RUNG wire#w1
      R_Coil( "reteaOut" )
   END_RUNG
   // the same network as SCL:
   #_w1 := "GVL"."STEP"[7] AND NOT "stare";
   IF #_w1 THEN
       "GVL"."STEP"[1] := TRUE;
       "GVL"."STEP"[7] := FALSE;
       "reteaOut" := FALSE;
   END_IF;
END_REGION

REGION Network 43: TR 8 - 4
   RUNG wire#powerrail
      Contact( "GVL"."STEP"[8] )
      Contact( "directieAuto" )
      { S7_Templates := "SrcType := Int" } GE_Contact(in1 := "Piata".PretPiata, in2 := "Piata".Prag)
      wire#w1
      S_Coil( "GVL"."STEP"[4] )
   END_RUNG
   RUNG wire#w1
      R_Coil( "GVL"."STEP"[8] )
   END_RUNG
   RUNG wire#w1
      R_Coil( "baterieOut" )
   END_RUNG
   // the same network as SCL:
   #_w1 := "GVL"."STEP"[8] AND "directieAuto" AND ("Piata".PretPiata >= "Piata".Prag);
   IF #_w1 THEN
       "GVL"."STEP"[4] := TRUE;
       "GVL"."STEP"[8] := FALSE;
       "baterieOut" := FALSE;
   END_IF;
END_REGION

REGION Network 44: TR 8 - 2
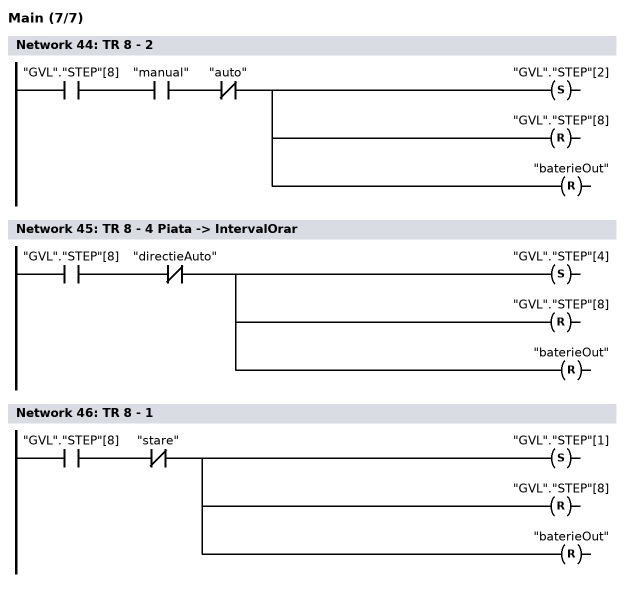
   RUNG wire#powerrail
      Contact( "GVL"."STEP"[8] )
      Contact( "manual" )
      I_Contact( "auto" )
      wire#w1
      S_Coil( "GVL"."STEP"[2] )
   END_RUNG
   RUNG wire#w1
      R_Coil( "GVL"."STEP"[8] )
   END_RUNG
   RUNG wire#w1
      R_Coil( "baterieOut" )
   END_RUNG
   // the same network as SCL:
   #_w1 := "GVL"."STEP"[8] AND "manual" AND NOT "auto";
   IF #_w1 THEN
       "GVL"."STEP"[2] := TRUE;
       "GVL"."STEP"[8] := FALSE;
       "baterieOut" := FALSE;
   END_IF;
END_REGION

REGION Network 45: TR 8 - 4 Piata -> IntervalOrar
   RUNG wire#powerrail
      Contact( "GVL"."STEP"[8] )
      I_Contact( "directieAuto" )
      wire#w1
      S_Coil( "GVL"."STEP"[4] )
   END_RUNG
   RUNG wire#w1
      R_Coil( "GVL"."STEP"[8] )
   END_RUNG
   RUNG wire#w1
      R_Coil( "baterieOut" )
   END_RUNG
   // the same network as SCL:
   #_w1 := "GVL"."STEP"[8] AND NOT "directieAuto";
   IF #_w1 THEN
       "GVL"."STEP"[4] := TRUE;
       "GVL"."STEP"[8] := FALSE;
       "baterieOut" := FALSE;
   END_IF;
END_REGION

REGION Network 46: TR 8 - 1
   RUNG wire#powerrail
      Contact( "GVL"."STEP"[8] )
      I_Contact( "stare" )
      wire#w1
      S_Coil( "GVL"."STEP"[1] )
   END_RUNG
   RUNG wire#w1
      R_Coil( "GVL"."STEP"[8] )
   END_RUNG
   RUNG wire#w1
      R_Coil( "baterieOut" )
   END_RUNG
   // the same network as SCL:
   #_w1 := "GVL"."STEP"[8] AND NOT "stare";
   IF #_w1 THEN
       "GVL"."STEP"[1] := TRUE;
       "GVL"."STEP"[8] := FALSE;
       "baterieOut" := FALSE;
   END_IF;
END_REGION
END_ORGANIZATION_BLOCK

ORGANIZATION_BLOCK "Modbus"   // OB123, LAD, ProgramCycle
TITLE = "Main Program Sweep (Cycle)"
{ S7_Optimized_Access := 'TRUE' }
VERSION : 0.1
   VAR_INPUT
      Initial_Call : Bool;   // Initial call of this OB
      Remanence : Bool;   // =True, if remanent data are available
   END_VAR
   VAR_TEMP   // added for the SCL form of the ladder/FBD networks
      _w1 : Bool;
      _w2 : Bool;
   END_VAR
BEGIN

REGION Network 1: "R_TRIG_Stare"
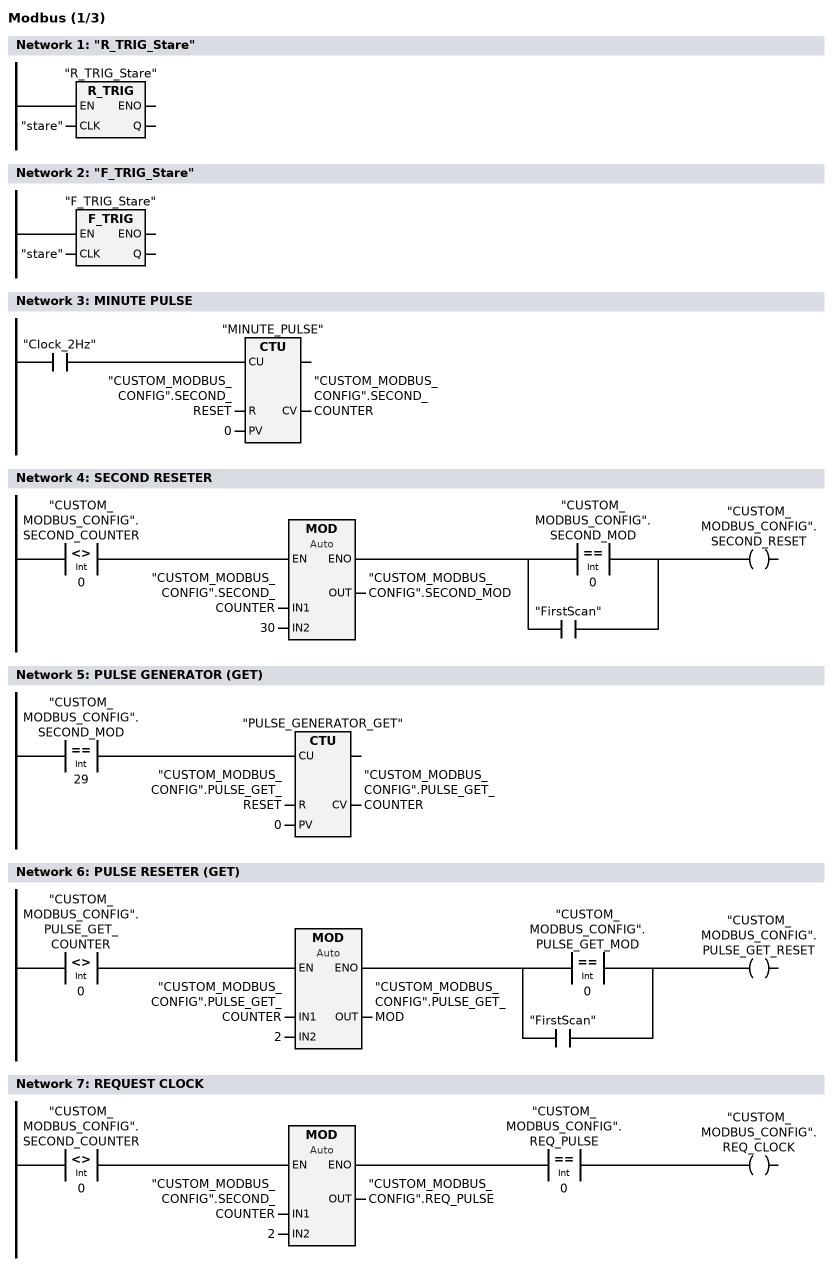
   "R_TRIG_Stare"(CLK := "stare");   // R_TRIG
END_REGION

REGION Network 2: "F_TRIG_Stare"
   "F_TRIG_Stare"(CLK := "stare");   // F_TRIG
END_REGION

REGION Network 3: MINUTE PULSE
   "MINUTE_PULSE".CTU(CU := "Clock_2Hz",
                      R := "CUSTOM_MODBUS_CONFIG".SECOND_RESET,
                      PV := 0,
                      CV => "CUSTOM_MODBUS_CONFIG".SECOND_COUNTER);
END_REGION

REGION Network 4: SECOND RESETER
   RUNG wire#powerrail
      { S7_Templates := "SrcType := Int" } NE_Contact(in1 := "CUSTOM_MODBUS_CONFIG".SECOND_COUNTER, in2 := 0)
      Mod(in1 := "CUSTOM_MODBUS_CONFIG".SECOND_COUNTER, in2 := 30, out => "CUSTOM_MODBUS_CONFIG".SECOND_MOD)
      wire#w1
      { S7_Templates := "SrcType := Int" } EQ_Contact(in1 := "CUSTOM_MODBUS_CONFIG".SECOND_MOD, in2 := 0)
      wire#w2
      Coil( "CUSTOM_MODBUS_CONFIG".SECOND_RESET )
   END_RUNG
   RUNG wire#w1
      Contact( "FirstScan" )
   END_RUNG wire#w2
   // the same network as SCL:
   #_w1 := "CUSTOM_MODBUS_CONFIG".SECOND_COUNTER <> 0;
   IF #_w1 THEN "CUSTOM_MODBUS_CONFIG".SECOND_MOD := "CUSTOM_MODBUS_CONFIG".SECOND_COUNTER MOD 30; END_IF;
   "CUSTOM_MODBUS_CONFIG".SECOND_RESET := #_w1 AND (("CUSTOM_MODBUS_CONFIG".SECOND_MOD = 0) OR "FirstScan");
END_REGION

REGION Network 5: PULSE GENERATOR (GET)
   "PULSE_GENERATOR_GET".CTU(CU := "CUSTOM_MODBUS_CONFIG".SECOND_MOD = 29,
                           R := "CUSTOM_MODBUS_CONFIG".PULSE_GET_RESET,
                           PV := 0,
                           CV => "CUSTOM_MODBUS_CONFIG".PULSE_GET_COUNTER);
END_REGION

REGION Network 6: PULSE RESETER (GET)
   RUNG wire#powerrail
      { S7_Templates := "SrcType := Int" } NE_Contact(in1 := "CUSTOM_MODBUS_CONFIG".PULSE_GET_COUNTER, in2 := 0)
      Mod(in1 := "CUSTOM_MODBUS_CONFIG".PULSE_GET_COUNTER, in2 := 2, out => "CUSTOM_MODBUS_CONFIG".PULSE_GET_MOD)
      wire#w1
      { S7_Templates := "SrcType := Int" } EQ_Contact(in1 := "CUSTOM_MODBUS_CONFIG".PULSE_GET_MOD, in2 := 0)
      wire#w2
      Coil( "CUSTOM_MODBUS_CONFIG".PULSE_GET_RESET )
   END_RUNG
   RUNG wire#w1
      Contact( "FirstScan" )
   END_RUNG wire#w2
   // the same network as SCL:
   #_w1 := "CUSTOM_MODBUS_CONFIG".PULSE_GET_COUNTER <> 0;
   IF #_w1 THEN
       "CUSTOM_MODBUS_CONFIG".PULSE_GET_MOD := "CUSTOM_MODBUS_CONFIG".PULSE_GET_COUNTER MOD 2;
   END_IF;
   "CUSTOM_MODBUS_CONFIG".PULSE_GET_RESET := #_w1 AND (("CUSTOM_MODBUS_CONFIG".PULSE_GET_MOD = 0) OR "FirstScan");
END_REGION

REGION Network 7: REQUEST CLOCK
   RUNG wire#powerrail
      { S7_Templates := "SrcType := Int" } NE_Contact(in1 := "CUSTOM_MODBUS_CONFIG".SECOND_COUNTER, in2 := 0)
      Mod(in1 := "CUSTOM_MODBUS_CONFIG".SECOND_COUNTER, in2 := 2, out => "CUSTOM_MODBUS_CONFIG".REQ_PULSE)
      { S7_Templates := "SrcType := Int" } EQ_Contact(in1 := "CUSTOM_MODBUS_CONFIG".REQ_PULSE, in2 := 0)
      Coil( "CUSTOM_MODBUS_CONFIG".REQ_CLOCK )
   END_RUNG
   // the same network as SCL:
   #_w1 := "CUSTOM_MODBUS_CONFIG".SECOND_COUNTER <> 0;
   IF #_w1 THEN "CUSTOM_MODBUS_CONFIG".REQ_PULSE := "CUSTOM_MODBUS_CONFIG".SECOND_COUNTER MOD 2; END_IF;
   "CUSTOM_MODBUS_CONFIG".REQ_CLOCK := #_w1 AND ("CUSTOM_MODBUS_CONFIG".REQ_PULSE = 0);
END_REGION

REGION Network 8: GET_CURR_HOUR_YIELD
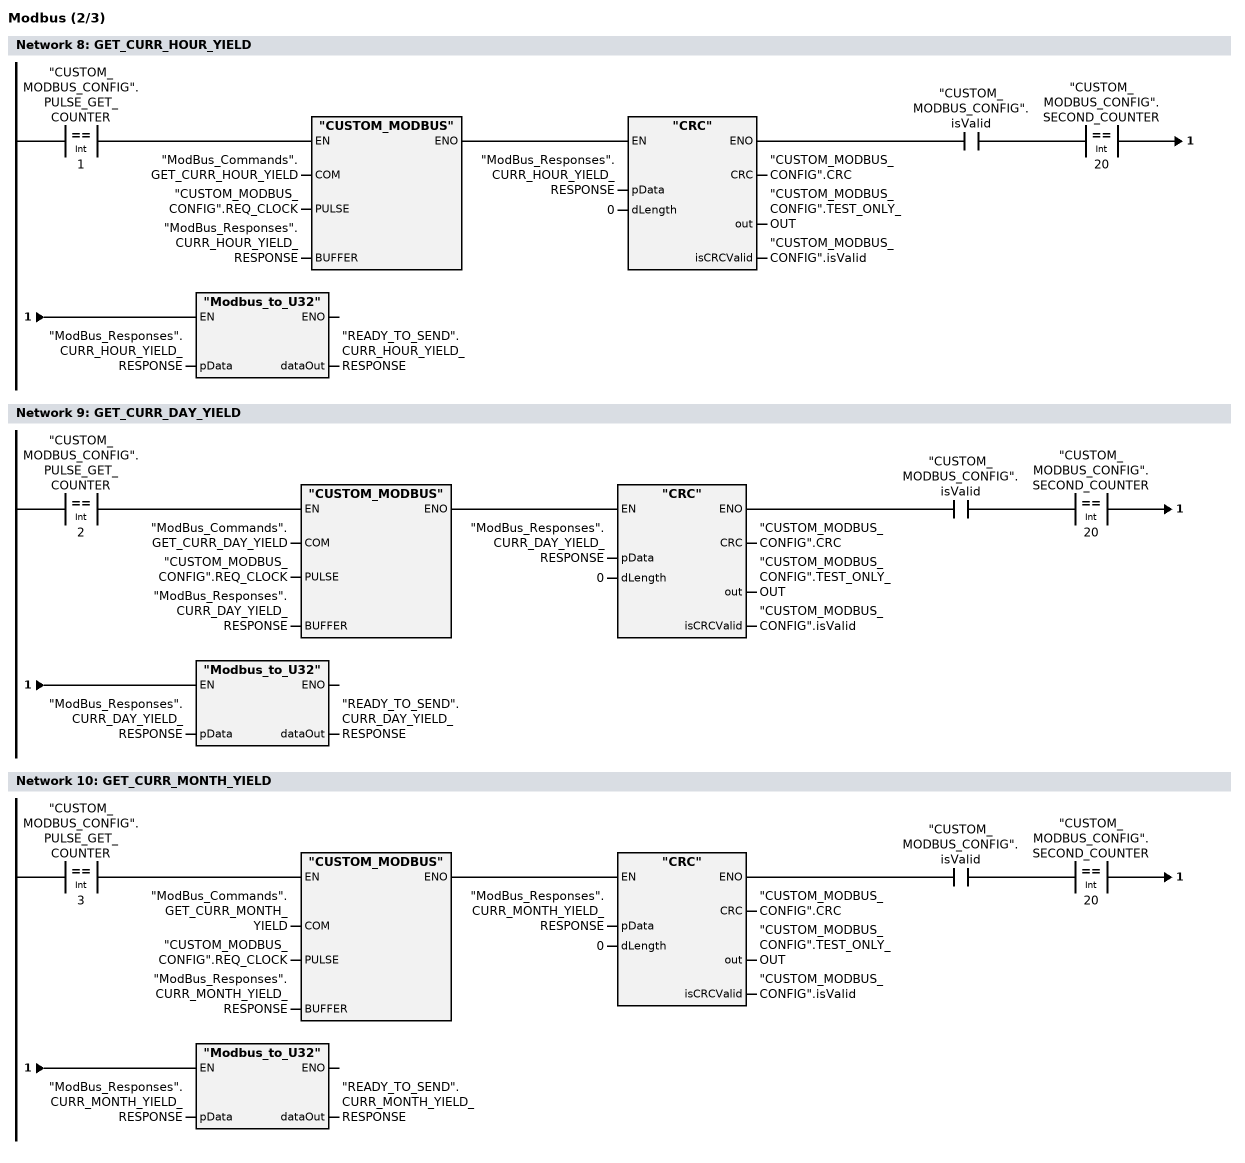
   RUNG wire#powerrail
      { S7_Templates := "SrcType := Int" } EQ_Contact(in1 := "CUSTOM_MODBUS_CONFIG".PULSE_GET_COUNTER, in2 := 1)
      "CUSTOM_MODBUS"(COM := "ModBus_Commands".GET_CURR_HOUR_YIELD, PULSE := "CUSTOM_MODBUS_CONFIG".REQ_CLOCK, BUFFER := "ModBus_Responses".CURR_HOUR_YIELD_RESPONSE)
      "CRC"(pData := "ModBus_Responses".CURR_HOUR_YIELD_RESPONSE, dLength := 0, CRC => "CUSTOM_MODBUS_CONFIG".CRC, out => "CUSTOM_MODBUS_CONFIG".TEST_ONLY_OUT, isCRCValid => "CUSTOM_MODBUS_CONFIG".isValid)
      Contact( "CUSTOM_MODBUS_CONFIG".isValid )
      { S7_Templates := "SrcType := Int" } EQ_Contact(in1 := "CUSTOM_MODBUS_CONFIG".SECOND_COUNTER, in2 := 20)
      "Modbus_to_U32"(pData := "ModBus_Responses".CURR_HOUR_YIELD_RESPONSE, dataOut => "READY_TO_SEND".CURR_HOUR_YIELD_RESPONSE)
   END_RUNG
   // the same network as SCL:
   "CUSTOM_MODBUS"(EN := "CUSTOM_MODBUS_CONFIG".PULSE_GET_COUNTER = 1,
                   COM := "ModBus_Commands".GET_CURR_HOUR_YIELD,
                   PULSE := "CUSTOM_MODBUS_CONFIG".REQ_CLOCK,
                   BUFFER := "ModBus_Responses".CURR_HOUR_YIELD_RESPONSE,
                   ENO => #_w1);
   "CRC"(EN := #_w1,
         pData := "ModBus_Responses".CURR_HOUR_YIELD_RESPONSE,
         dLength := 0,
         CRC => "CUSTOM_MODBUS_CONFIG".CRC,
         out => "CUSTOM_MODBUS_CONFIG".TEST_ONLY_OUT,
         isCRCValid => "CUSTOM_MODBUS_CONFIG".isValid,
         ENO => #_w2);
   IF #_w2 AND "CUSTOM_MODBUS_CONFIG".isValid AND ("CUSTOM_MODBUS_CONFIG".SECOND_COUNTER = 20) THEN
       "Modbus_to_U32"(pData := "ModBus_Responses".CURR_HOUR_YIELD_RESPONSE,
                       dataOut => "READY_TO_SEND".CURR_HOUR_YIELD_RESPONSE);
   END_IF;
END_REGION

REGION Network 9: GET_CURR_DAY_YIELD
   RUNG wire#powerrail
      { S7_Templates := "SrcType := Int" } EQ_Contact(in1 := "CUSTOM_MODBUS_CONFIG".PULSE_GET_COUNTER, in2 := 2)
      "CUSTOM_MODBUS"(COM := "ModBus_Commands".GET_CURR_DAY_YIELD, PULSE := "CUSTOM_MODBUS_CONFIG".REQ_CLOCK, BUFFER := "ModBus_Responses".CURR_DAY_YIELD_RESPONSE)
      "CRC"(pData := "ModBus_Responses".CURR_DAY_YIELD_RESPONSE, dLength := 0, CRC => "CUSTOM_MODBUS_CONFIG".CRC, out => "CUSTOM_MODBUS_CONFIG".TEST_ONLY_OUT, isCRCValid => "CUSTOM_MODBUS_CONFIG".isValid)
      Contact( "CUSTOM_MODBUS_CONFIG".isValid )
      { S7_Templates := "SrcType := Int" } EQ_Contact(in1 := "CUSTOM_MODBUS_CONFIG".SECOND_COUNTER, in2 := 20)
      "Modbus_to_U32"(pData := "ModBus_Responses".CURR_DAY_YIELD_RESPONSE, dataOut => "READY_TO_SEND".CURR_DAY_YIELD_RESPONSE)
   END_RUNG
   // the same network as SCL:
   "CUSTOM_MODBUS"(EN := "CUSTOM_MODBUS_CONFIG".PULSE_GET_COUNTER = 2,
                   COM := "ModBus_Commands".GET_CURR_DAY_YIELD,
                   PULSE := "CUSTOM_MODBUS_CONFIG".REQ_CLOCK,
                   BUFFER := "ModBus_Responses".CURR_DAY_YIELD_RESPONSE,
                   ENO => #_w1);
   "CRC"(EN := #_w1,
         pData := "ModBus_Responses".CURR_DAY_YIELD_RESPONSE,
         dLength := 0,
         CRC => "CUSTOM_MODBUS_CONFIG".CRC,
         out => "CUSTOM_MODBUS_CONFIG".TEST_ONLY_OUT,
         isCRCValid => "CUSTOM_MODBUS_CONFIG".isValid,
         ENO => #_w2);
   IF #_w2 AND "CUSTOM_MODBUS_CONFIG".isValid AND ("CUSTOM_MODBUS_CONFIG".SECOND_COUNTER = 20) THEN
       "Modbus_to_U32"(pData := "ModBus_Responses".CURR_DAY_YIELD_RESPONSE,
                       dataOut => "READY_TO_SEND".CURR_DAY_YIELD_RESPONSE);
   END_IF;
END_REGION

REGION Network 10: GET_CURR_MONTH_YIELD
   RUNG wire#powerrail
      { S7_Templates := "SrcType := Int" } EQ_Contact(in1 := "CUSTOM_MODBUS_CONFIG".PULSE_GET_COUNTER, in2 := 3)
      "CUSTOM_MODBUS"(COM := "ModBus_Commands".GET_CURR_MONTH_YIELD, PULSE := "CUSTOM_MODBUS_CONFIG".REQ_CLOCK, BUFFER := "ModBus_Responses".CURR_MONTH_YIELD_RESPONSE)
      "CRC"(pData := "ModBus_Responses".CURR_MONTH_YIELD_RESPONSE, dLength := 0, CRC => "CUSTOM_MODBUS_CONFIG".CRC, out => "CUSTOM_MODBUS_CONFIG".TEST_ONLY_OUT, isCRCValid => "CUSTOM_MODBUS_CONFIG".isValid)
      Contact( "CUSTOM_MODBUS_CONFIG".isValid )
      { S7_Templates := "SrcType := Int" } EQ_Contact(in1 := "CUSTOM_MODBUS_CONFIG".SECOND_COUNTER, in2 := 20)
      "Modbus_to_U32"(pData := "ModBus_Responses".CURR_MONTH_YIELD_RESPONSE, dataOut => "READY_TO_SEND".CURR_MONTH_YIELD_RESPONSE)
   END_RUNG
   // the same network as SCL:
   "CUSTOM_MODBUS"(EN := "CUSTOM_MODBUS_CONFIG".PULSE_GET_COUNTER = 3,
                   COM := "ModBus_Commands".GET_CURR_MONTH_YIELD,
                   PULSE := "CUSTOM_MODBUS_CONFIG".REQ_CLOCK,
                   BUFFER := "ModBus_Responses".CURR_MONTH_YIELD_RESPONSE,
                   ENO => #_w1);
   "CRC"(EN := #_w1,
         pData := "ModBus_Responses".CURR_MONTH_YIELD_RESPONSE,
         dLength := 0,
         CRC => "CUSTOM_MODBUS_CONFIG".CRC,
         out => "CUSTOM_MODBUS_CONFIG".TEST_ONLY_OUT,
         isCRCValid => "CUSTOM_MODBUS_CONFIG".isValid,
         ENO => #_w2);
   IF #_w2 AND "CUSTOM_MODBUS_CONFIG".isValid AND ("CUSTOM_MODBUS_CONFIG".SECOND_COUNTER = 20) THEN
       "Modbus_to_U32"(pData := "ModBus_Responses".CURR_MONTH_YIELD_RESPONSE,
                       dataOut => "READY_TO_SEND".CURR_MONTH_YIELD_RESPONSE);
   END_IF;
END_REGION

REGION Network 11: GET_DEVICE_STATUS
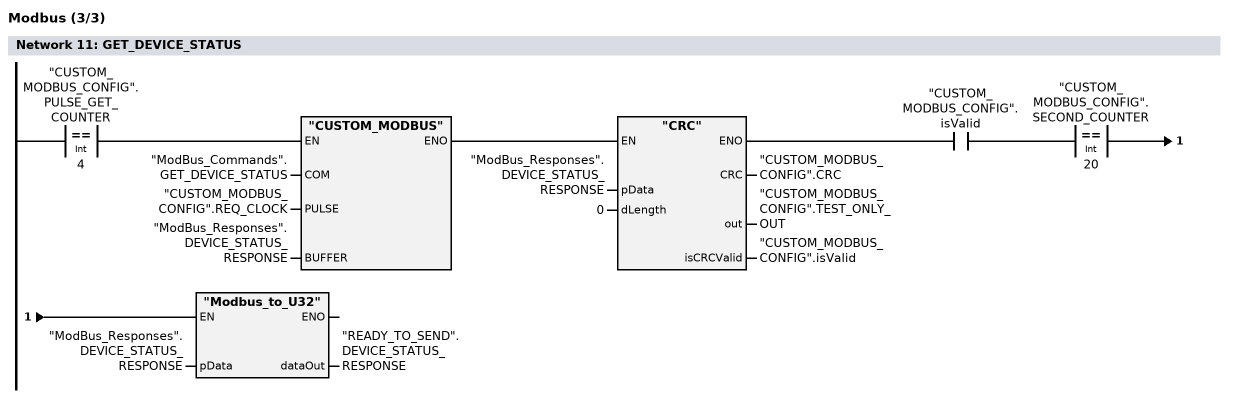
   RUNG wire#powerrail
      { S7_Templates := "SrcType := Int" } EQ_Contact(in1 := "CUSTOM_MODBUS_CONFIG".PULSE_GET_COUNTER, in2 := 4)
      "CUSTOM_MODBUS"(COM := "ModBus_Commands".GET_DEVICE_STATUS, PULSE := "CUSTOM_MODBUS_CONFIG".REQ_CLOCK, BUFFER := "ModBus_Responses".DEVICE_STATUS_RESPONSE)
      "CRC"(pData := "ModBus_Responses".DEVICE_STATUS_RESPONSE, dLength := 0, CRC => "CUSTOM_MODBUS_CONFIG".CRC, out => "CUSTOM_MODBUS_CONFIG".TEST_ONLY_OUT, isCRCValid => "CUSTOM_MODBUS_CONFIG".isValid)
      Contact( "CUSTOM_MODBUS_CONFIG".isValid )
      { S7_Templates := "SrcType := Int" } EQ_Contact(in1 := "CUSTOM_MODBUS_CONFIG".SECOND_COUNTER, in2 := 20)
      "Modbus_to_U32"(pData := "ModBus_Responses".DEVICE_STATUS_RESPONSE, dataOut => "READY_TO_SEND".DEVICE_STATUS_RESPONSE)
   END_RUNG
   // the same network as SCL:
   "CUSTOM_MODBUS"(EN := "CUSTOM_MODBUS_CONFIG".PULSE_GET_COUNTER = 4,
                   COM := "ModBus_Commands".GET_DEVICE_STATUS,
                   PULSE := "CUSTOM_MODBUS_CONFIG".REQ_CLOCK,
                   BUFFER := "ModBus_Responses".DEVICE_STATUS_RESPONSE,
                   ENO => #_w1);
   "CRC"(EN := #_w1,
         pData := "ModBus_Responses".DEVICE_STATUS_RESPONSE,
         dLength := 0,
         CRC => "CUSTOM_MODBUS_CONFIG".CRC,
         out => "CUSTOM_MODBUS_CONFIG".TEST_ONLY_OUT,
         isCRCValid => "CUSTOM_MODBUS_CONFIG".isValid,
         ENO => #_w2);
   IF #_w2 AND "CUSTOM_MODBUS_CONFIG".isValid AND ("CUSTOM_MODBUS_CONFIG".SECOND_COUNTER = 20) THEN
       "Modbus_to_U32"(pData := "ModBus_Responses".DEVICE_STATUS_RESPONSE,
                       dataOut => "READY_TO_SEND".DEVICE_STATUS_RESPONSE);
   END_IF;
END_REGION
END_ORGANIZATION_BLOCK

ORGANIZATION_BLOCK "get_time"   // OB124, LAD, ProgramCycle
TITLE = "Main Program Sweep (Cycle)"
{ S7_Optimized_Access := 'TRUE' }
VERSION : 0.1
   VAR_INPUT
      Initial_Call : Bool;   // Initial call of this OB
      Remanence : Bool;   // =True, if remanent data are available
   END_VAR
BEGIN

REGION Network 1
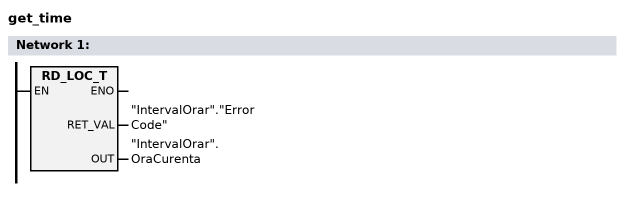
   "IntervalOrar"."Error Code" := RD_LOC_T(OUT => "IntervalOrar".OraCurenta);
END_REGION
END_ORGANIZATION_BLOCK

ORGANIZATION_BLOCK "Modbus_Logic"   // OB125, LAD, ProgramCycle
TITLE = "Main Program Sweep (Cycle)"
{ S7_Optimized_Access := 'TRUE' }
VERSION : 0.1
   VAR_INPUT
      Initial_Call : Bool;   // Initial call of this OB
      Remanence : Bool;   // =True, if remanent data are available
   END_VAR
   VAR_TEMP   // added for the SCL form of the ladder/FBD networks
      _w1 : Bool;
   END_VAR
BEGIN

REGION Network 1: PULSE GENERATOR (SET)
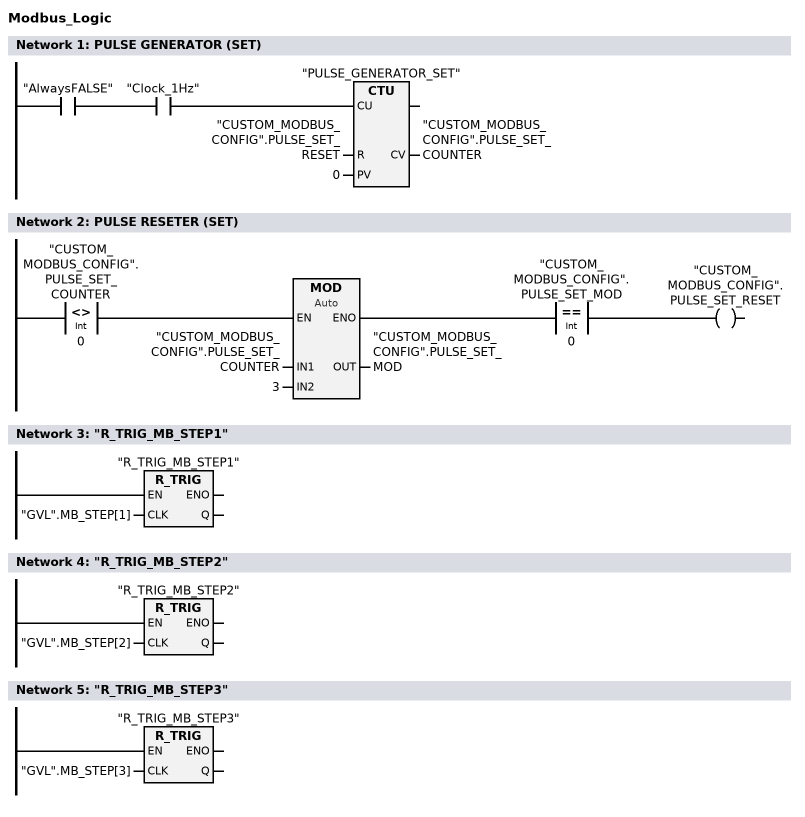
   "PULSE_GENERATOR_SET".CTU(CU := "AlwaysFALSE" AND "Clock_1Hz",
                           R := "CUSTOM_MODBUS_CONFIG".PULSE_SET_RESET,
                           PV := 0,
                           CV => "CUSTOM_MODBUS_CONFIG".PULSE_SET_COUNTER);
END_REGION

REGION Network 2: PULSE RESETER (SET)
   RUNG wire#powerrail
      { S7_Templates := "SrcType := Int" } NE_Contact(in1 := "CUSTOM_MODBUS_CONFIG".PULSE_SET_COUNTER, in2 := 0)
      Mod(in1 := "CUSTOM_MODBUS_CONFIG".PULSE_SET_COUNTER, in2 := 3, out => "CUSTOM_MODBUS_CONFIG".PULSE_SET_MOD)
      { S7_Templates := "SrcType := Int" } EQ_Contact(in1 := "CUSTOM_MODBUS_CONFIG".PULSE_SET_MOD, in2 := 0)
      Coil( "CUSTOM_MODBUS_CONFIG".PULSE_SET_RESET )
   END_RUNG
   // the same network as SCL:
   #_w1 := "CUSTOM_MODBUS_CONFIG".PULSE_SET_COUNTER <> 0;
   IF #_w1 THEN
       "CUSTOM_MODBUS_CONFIG".PULSE_SET_MOD := "CUSTOM_MODBUS_CONFIG".PULSE_SET_COUNTER MOD 3;
   END_IF;
   "CUSTOM_MODBUS_CONFIG".PULSE_SET_RESET := #_w1 AND ("CUSTOM_MODBUS_CONFIG".PULSE_SET_MOD = 0);
END_REGION

REGION Network 3: "R_TRIG_MB_STEP1"
   "R_TRIG_MB_STEP1"(CLK := "GVL".MB_STEP[1]);   // R_TRIG
END_REGION

REGION Network 4: "R_TRIG_MB_STEP2"
   "R_TRIG_MB_STEP2"(CLK := "GVL".MB_STEP[2]);   // R_TRIG
END_REGION

REGION Network 5: "R_TRIG_MB_STEP3"
   "R_TRIG_MB_STEP3"(CLK := "GVL".MB_STEP[3]);   // R_TRIG
END_REGION
END_ORGANIZATION_BLOCK

ORGANIZATION_BLOCK "send_to_server"   // OB126, LAD, ProgramCycle
TITLE = "Main Program Sweep (Cycle)"
{ S7_Optimized_Access := 'TRUE' }
VERSION : 0.1
   VAR_INPUT
      Initial_Call : Bool;   // Initial call of this OB
      Remanence : Bool;   // =True, if remanent data are available
   END_VAR
BEGIN

REGION Network 1
   // IN POZITIA 0 A CICLULUI DE COMEZI TRIMIT TOATE DATELE DIN READY_TO_SEND SPRE SERVER
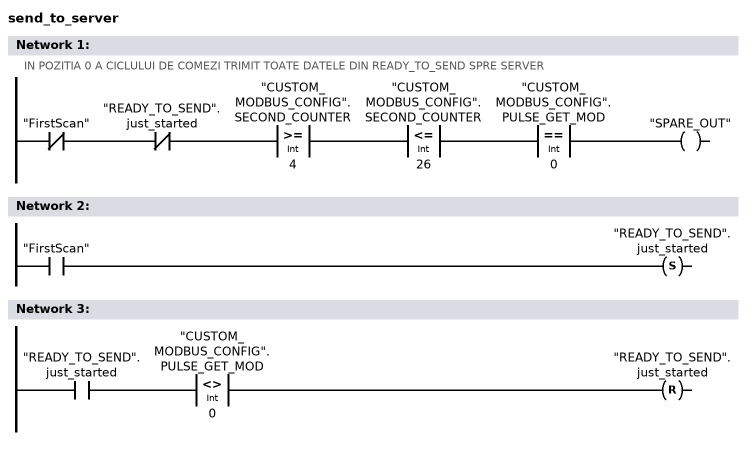
   RUNG wire#powerrail
      I_Contact( "FirstScan" )
      I_Contact( "READY_TO_SEND".just_started )
      { S7_Templates := "SrcType := Int" } GE_Contact(in1 := "CUSTOM_MODBUS_CONFIG".SECOND_COUNTER, in2 := 4)
      { S7_Templates := "SrcType := Int" } LE_Contact(in1 := "CUSTOM_MODBUS_CONFIG".SECOND_COUNTER, in2 := 26)
      { S7_Templates := "SrcType := Int" } EQ_Contact(in1 := "CUSTOM_MODBUS_CONFIG".PULSE_GET_MOD, in2 := 0)
      Coil( "SPARE_OUT" )
   END_RUNG
   // the same network as SCL:
   "SPARE_OUT" := NOT "FirstScan" AND NOT "READY_TO_SEND".just_started AND ("CUSTOM_MODBUS_CONFIG".SECOND_COUNTER >= 4) AND ("CUSTOM_MODBUS_CONFIG".SECOND_COUNTER <= 26) AND ("CUSTOM_MODBUS_CONFIG".PULSE_GET_MOD = 0);
END_REGION

REGION Network 2
   RUNG wire#powerrail
      Contact( "FirstScan" )
      S_Coil( "READY_TO_SEND".just_started )
   END_RUNG
   // the same network as SCL:
   IF "FirstScan" THEN "READY_TO_SEND".just_started := TRUE; END_IF;
END_REGION

REGION Network 3
   RUNG wire#powerrail
      Contact( "READY_TO_SEND".just_started )
      { S7_Templates := "SrcType := Int" } NE_Contact(in1 := "CUSTOM_MODBUS_CONFIG".PULSE_GET_MOD, in2 := 0)
      R_Coil( "READY_TO_SEND".just_started )
   END_RUNG
   // the same network as SCL:
   IF "READY_TO_SEND".just_started AND ("CUSTOM_MODBUS_CONFIG".PULSE_GET_MOD <> 0) THEN
       "READY_TO_SEND".just_started := FALSE;
   END_IF;
END_REGION
END_ORGANIZATION_BLOCK